# B&R Automation Studio project GAT (part 9)

#### CamAutomatActions.st
```iecst
//*********************************************************************************
//* Copyright: B&R Industrial Automation GmbH
//* Author:    B&R Industrial Automation GmbH
//* Created:   24 June, 2021/15:05
//* This task reads the cam automat data from the ACOPOS into the PV structure
//*********************************************************************************

ACTION InitCamAutFunctionBlocks:
	// Init cam automat related function blocks
	McCamAutDefine.DataAddress := ADR(McCamAutPar);
	MC_BR_CamAutomatGetPar_AcpAx_0.Slave := ADR(gAxisSlave);
	MC_BR_CamAutomatGetPar_AcpAx_0.Command := mcGET_PAR_ACTUAL;
	MC_BR_CamAutomatGetPar_AcpAx_0.CamAutomat := McCamAutDefine;
    MC_BR_CamAutomatSetPar_AcpAx_0.Command := mcSET_UPDATE_FROM_ADR;
    // Synchron means the new parameters are valid when an event with synchronous update = TRUE happens
	MC_BR_CamAutomatSetPar_AcpAx_0.AdvancedParameters.ParLock := mcCAMAUT_UNLOCK_SYNCHRON;
	MC_BR_CamAutomatSetPar_AcpAx_0.CamAutomat := McCamAutDefine;
	MC_BR_CamAutomatSetPar_AcpAx_0.Slave := ADR(gAxisSlave);
	MC_BR_CamAutomatCommand_0.Slave := ADR(gAxisSlave);
	MC_BR_CamAutomatCommand_0.Enable := TRUE;
END_ACTION

ACTION GetCamAutPar:
	CASE InitCamAut OF
		0: // Set up function blocks for reading and writing cam automat parameters
			MC_BR_CamAutomatGetPar_AcpAx_0.Execute := TRUE;
			InitCamAut := 1;

		1: // Wait for function block done
			IF MC_BR_CamAutomatGetPar_AcpAx_0.Done THEN
				MC_BR_CamAutomatGetPar_AcpAx_0.Execute := FALSE;
				InitCamAut := 10;
			END_IF
			// In case of error abort reading
			IF MC_BR_CamAutomatGetPar_AcpAx_0.Error THEN
				MC_BR_CamAutomatGetPar_AcpAx_0.Execute := FALSE;
				InitCamAut := 100;
			END_IF

		10: // Done, do nothing

		100: // Error handling
	END_CASE;
END_ACTION

ACTION UpdateCamAutomatAction:
	CASE CamUpdateState OF
		0: // Calculate new cam automat parameters
			IF UpdateCamAutomat AND (InitCamAut = 10) THEN
				// General CAM settings
				McCamAutPar.Common.Master.MasterStartInterval := MainCtrl.Intern.ProductLength[MainCtrl.Status.CurrentBatch];
				McCamAutPar.Common.Master.MasterStartPosition := 0;

				// CAM state 0: Base state, wait for master start position
				McCamAutPar.State[0].Event[0].NextState := 1;
				McCamAutPar.State[0].Event[0].SynchronousUpdate := mcSWITCH_ON;
                McCamAutPar.State[0].Event[0].Transition := mcEVENT_IMMEDIATELY;
                // Starts cutting process on interval, modify according to machine e.g. change to mcEVENT_SRC_TRIGGER1 for a signal wired to input channel 1 on ACOPOS
				McCamAutPar.State[0].Event[0].Type := mcEVENT_START_POSITION;

                // CAM state 1: First cut movement
                // * 100 because of measurement units to resolution units conversion
                McCamAutPar.State[1].MasterFactor := REAL_TO_DINT(GatDegreeToDistance(MainCtrl.FixParameter.SyncAngle, MainCtrl.FixParameter.CutDiameter / 2) * 100);
                // * 100 because of measurement units to resolution units conversion
                McCamAutPar.State[1].SlaveFactor := REAL_TO_DINT(MainCtrl.FixParameter.SyncAngle * 100);
                // Assuming print mark signals coincide with cutting positions
				McCamAutPar.State[1].CompensationParameters.MasterCompDistance := MainCtrl.Intern.ProductLength[MainCtrl.Status.CurrentBatch];
				IF MainCtrl.FixParameter.NrOfKnives = 0 THEN
					// There must be at least one knife!
					MainCtrl.FixParameter.NrOfKnives := 1;
				END_IF
				McCamAutPar.State[1].CompensationParameters.SlaveCompDistance := (360 / (2 * MainCtrl.FixParameter.NrOfKnives)) - (MainCtrl.FixParameter.SyncAngle / 2);
				// Change to next state at end of state
				McCamAutPar.State[1].Event[0].NextState := 3;
				McCamAutPar.State[1].Event[0].SynchronousUpdate := mcSWITCH_ON;
				McCamAutPar.State[1].Event[0].Transition := mcEVENT_END_OF_STATE;
				McCamAutPar.State[1].Event[0].Type := mcEVENT_SIGNAL2;
				McCamAutPar.State[1].Event[1].NextState := 2;
				McCamAutPar.State[1].Event[1].SynchronousUpdate := mcSWITCH_ON;
				McCamAutPar.State[1].Event[1].Transition := mcEVENT_END_OF_STATE;
				McCamAutPar.State[1].Event[1].Type := mcEVENT_STATE_END;

                // CAM state 2: Repeating cut movements
                // * 100 because of measurement units to resolution units conversion
				McCamAutPar.State[2].MasterFactor := REAL_TO_DINT(GatDegreeToDistance(MainCtrl.FixParameter.SyncAngle, MainCtrl.FixParameter.CutDiameter / 2) * 100);
				McCamAutPar.State[2].SlaveFactor := REAL_TO_DINT(MainCtrl.FixParameter.SyncAngle * 100);// * 100 because of measurement units to resolution units conversion
				McCamAutPar.State[2].CompensationParameters.MasterCompDistance := MainCtrl.Intern.ProductLength[MainCtrl.Status.CurrentBatch];
				McCamAutPar.State[2].CompensationParameters.SlaveCompDistance := (360 / MainCtrl.FixParameter.NrOfKnives);
				// Repeat state at end of state, or go to next state in case of signal 2 (stop cutting signal)
				McCamAutPar.State[2].Event[0].NextState := 3;
				McCamAutPar.State[2].Event[0].SynchronousUpdate := mcSWITCH_ON;
				McCamAutPar.State[2].Event[0].Transition := mcEVENT_END_OF_STATE;
				McCamAutPar.State[2].Event[0].Type := mcEVENT_SIGNAL2;
				McCamAutPar.State[2].Event[1].NextState := 2;
				McCamAutPar.State[2].Event[1].SynchronousUpdate := mcSWITCH_ON;
				McCamAutPar.State[2].Event[1].Transition := mcEVENT_END_OF_STATE;
				McCamAutPar.State[2].Event[1].Type := mcEVENT_STATE_END;

                // CAM state 3: Decelerate and stop at home position
                // Master with any positive value & slave = 0 means slave is not moving
                McCamAutPar.State[3].MasterFactor := 100;
                // Master with any positive value & slave = 0 means slave is not moving
                McCamAutPar.State[3].SlaveFactor := 0;
                // allow half a product length to stop
				McCamAutPar.State[3].CompensationParameters.MasterCompDistance := MainCtrl.Intern.ProductLength[MainCtrl.Status.CurrentBatch] / 2;
				McCamAutPar.State[3].CompensationParameters.SlaveCompDistance := (360 / (2 * MainCtrl.FixParameter.NrOfKnives));
				// Return to base state after axis has stopped
				McCamAutPar.State[3].Event[0].NextState := 0;
				McCamAutPar.State[3].Event[0].SynchronousUpdate := mcSWITCH_ON;
				McCamAutPar.State[3].Event[0].Transition := mcEVENT_END_OF_STATE;
				McCamAutPar.State[3].Event[0].Type := mcEVENT_STATE_END;

				MC_BR_CamAutomatSetPar_AcpAx_0.Execute := TRUE;
				CamUpdateState := 1;
			END_IF

		1: // Wait for SetPar done
			IF MC_BR_CamAutomatSetPar_AcpAx_0.Done THEN
				UpdateCamAutomat := FALSE;
				MC_BR_CamAutomatSetPar_AcpAx_0.Execute := FALSE;
				CamUpdateState := 0;
			ELSIF MC_BR_CamAutomatSetPar_AcpAx_0.Error THEN
				// Error handling
				MpAlarmXSet(gMpLinkAlarmXCore, 'SetCamFailed');
				UpdateCamAutomat := FALSE;
				MC_BR_CamAutomatSetPar_AcpAx_0.Execute := FALSE;
				CamUpdateState := 0;
			END_IF
	END_CASE;
END_ACTION
```

#### CrossCutter.st
```iecst
//*********************************************************************************
//* Copyright: B&R Industrial Automation GmbH
//* Created:   29 June, 2021/10:43
//* Process specific logic to update production information and process parameters
//*********************************************************************************

ACTION CrossCutter:

	//****************************Starting and stopping the process*********************************
    IF MainCtrl.Command.AutoModeOn THEN
        // Switch on axes
		AxisControl[AXIS_IDX_FEEDER].Command.Power := TRUE;
		AxisControl[AXIS_IDX_CUTTER].Command.Power := TRUE;
		// Home axes if not homed yet
		IF NOT MpAxisBasic_x[AXIS_IDX_FEEDER].IsHomed AND (AxisControl[AXIS_IDX_FEEDER].AxisState = AX_STATE_WAIT) THEN
			AxisControl[AXIS_IDX_FEEDER].Command.Home := TRUE;
		END_IF
		IF NOT MpAxisBasic_x[AXIS_IDX_CUTTER].IsHomed AND (AxisControl[AXIS_IDX_CUTTER].AxisState = AX_STATE_WAIT) THEN
			AxisControl[AXIS_IDX_CUTTER].Command.Home := TRUE;
		END_IF

		// Reset run switches when in error state
		IF (AxisControl[AXIS_IDX_FEEDER].AxisState = AX_STATE_ERROR) OR (AxisControl[AXIS_IDX_CUTTER].AxisState = AX_STATE_ERROR) THEN
			MainCtrl.Command.RunCutter := FALSE;
			MainCtrl.Command.RunFeeder := FALSE;
		END_IF

		// Start movement of feeder axis
		AxisControl[AXIS_IDX_FEEDER].Command.MoveVelocity := MainCtrl.Command.RunFeeder;

		// Start synchronized movement of Cutter with cam automat
		IF MainCtrl.Command.RunCutter THEN
			AxisControl[AXIS_IDX_CUTTER].Command.RunCamAutomat := TRUE;
		ELSE
			// If axis is moving use signal1 to stop slave in home position after the current product is done, otherwise stop now
			IF (MpAxisBasic_x[AXIS_IDX_CUTTER].Velocity > 0) AND MC_BR_CamAutomatCommand_0.Running THEN
				MC_BR_CamAutomatCommand_0.SetSignal1 := TRUE;
			ELSE
				// Back in base state reset signal and end camautomat
				MC_BR_CamAutomatCommand_0.SetSignal1 := FALSE;
				MC_BR_CamAutomatCommand_0.EndAutomat := MC_BR_CamAutomatCommand_0.Running;
				IF NOT MC_BR_CamAutomatCommand_0.Running THEN
					// Automat has stopped
					AxisControl[AXIS_IDX_CUTTER].Command.RunCamAutomat := FALSE;
				END_IF
			END_IF
		END_IF
	ELSIF LastAutoModeOn THEN
		// Auto mode is switched off, reste run commands
		MainCtrl.Command.RunCutter := FALSE;
		AxisControl[AXIS_IDX_CUTTER].Command.RunCamAutomat := FALSE;
		MainCtrl.Command.RunFeeder := FALSE;
		AxisControl[AXIS_IDX_FEEDER].Command.MoveVelocity := FALSE;
	END_IF
	LastAutoModeOn := MainCtrl.Command.AutoModeOn;

	//********************************Parameters Limits************

	IF (AxisControl[AXIS_IDX_FEEDER].Parameter.AxPar.Velocity = 0) AND AxisControl[AXIS_IDX_FEEDER].Command.MoveVelocity THEN
		MpAlarmXSet(gMpLinkAlarmXCore, 'FeederSpeedNotSet');
		AxisControl[AXIS_IDX_FEEDER].Command.MoveVelocity := FALSE;
	END_IF
	IF (AxisControl[AXIS_IDX_CUTTER].Parameter.AxPar.Velocity = 0) AND AxisControl[AXIS_IDX_CUTTER].Command.MoveAdditive THEN
		MpAlarmXSet(gMpLinkAlarmXCore, 'CutterSpeedNotSet');
		AxisControl[AXIS_IDX_CUTTER].Command.MoveAdditive := FALSE;
	END_IF
	IF (AxisControl[AXIS_IDX_CUTTER].Parameter.AxPar.Distance = 0) AND (AxisControl[AXIS_IDX_CUTTER].Command.MoveAdditive)  THEN
		MpAlarmXSet(gMpLinkAlarmXCore, 'CutterPositionNotSet');
		AxisControl[AXIS_IDX_CUTTER].Command.MoveAdditive := FALSE;
	END_IF

	//****************************Product Cutting numbering*********************************
    // Update parameters on recipe load
    IF MpRecipeRegPar_P.UpdateNotification THEN
		brsmemcpy(ADR(MainCtrl.Intern.ProductLength), ADR(MainCtrl.Parameter.ProductLength), SIZEOF(MainCtrl.Intern.ProductLength));
		brsmemcpy(ADR(MainCtrl.Intern.ProductNumber), ADR(MainCtrl.Parameter.ProductNumber), SIZEOF(MainCtrl.Intern.ProductNumber));
		UpdateCamAutomat := TRUE;
	END_IF

	// InCam -> next cut is starting
	IF EDGEPOS(MC_BR_CamAutomatCommand_0.InCam) THEN
		MainCtrl.Status.ProductsCutBatch := MainCtrl.Status.ProductsCutBatch + 1;
		MainCtrl.Status.ProductsCutTotal := MainCtrl.Status.ProductsCutTotal + 1;
	END_IF

	// Batch finished, start next batch -> adjust cam automat parameters for next batches product length
	IF (MainCtrl.Status.ProductsCutBatch >= MainCtrl.Intern.ProductNumber[MainCtrl.Status.CurrentBatch])
		AND (MainCtrl.Status.ProductsCutBatch > 0) THEN
		// Set new cam automat values
		MainCtrl.Status.CurrentBatch := MainCtrl.Status.CurrentBatch + 1;
		IF MainCtrl.Status.CurrentBatch > 4 THEN
			MainCtrl.Status.CurrentBatch := 0;
		END_IF
		MainCtrl.Status.ProductsCutBatch := 0;
		UpdateCamAutomat := TRUE;
	END_IF
	MainCtrl.Status.CurrentBatchTarget := MainCtrl.Intern.ProductNumber[MainCtrl.Status.CurrentBatch];
	MainCtrl.Status.CurrentBatchLength := MainCtrl.Intern.ProductLength[MainCtrl.Status.CurrentBatch];

	// Action to handle cam automat updates
	UpdateCamAutomatAction;

END_ACTION
```

#### Main.st
```iecst
//*********************************************************************************
//* Copyright: B&R Industrial Automation GmbH
//* Author:    B&R Industrial Automation GmbH
//* Created:   30. Sep 2020/08:00
//* Description: Tasks for axis control. The Main Cross Cutter handling is done in this task.
//*********************************************************************************

PROGRAM _INIT
	// Register parameters to MpRecipe
	MpRecipeRegPar_M.MpLink := ADR(gMpLinkRecipeXml);
	MpRecipeRegPar_M.Enable := TRUE;
	MpRecipeRegPar_M.Category := ADR('Machine');
	MpRecipeRegPar_M.PVName := ADR('MainCtrl:MainCtrl.FixPar');
	MpRecipeRegPar_P.MpLink := ADR(gMpLinkRecipeXml);
	MpRecipeRegPar_P.Enable := TRUE;
	MpRecipeRegPar_P.Category := ADR('Parameters');
	MpRecipeRegPar_P.PVName := ADR('MainCtrl:MainCtrl.Para');
	MpRecipeRegPar_Pre1.MpLink := ADR(gRecipeXmlPreviewMpLink);
	MpRecipeRegPar_Pre1.Enable := TRUE;
	MpRecipeRegPar_Pre1.Category := ADR('Preview');
	MpRecipeRegPar_Pre1.PVName := ADR('MainCtrl:PreviewParameters');
	MpRecipeRegPar_Pre2.MpLink := ADR(gMpLinkRecipeXml);
	MpRecipeRegPar_Pre2.Enable := TRUE;
	MpRecipeRegPar_Pre2.Category := ADR('Parameters');
	MpRecipeRegPar_Pre2.PVName := ADR('MainCtrl:PreviewParameters');

	// Activate RegPar FUBs
	WHILE NOT MpRecipeRegPar_M.Active DO
		MpRecipeRegPar_M();
	END_WHILE
	WHILE NOT MpRecipeRegPar_P.Active DO
		MpRecipeRegPar_P();
	END_WHILE
	WHILE NOT MpRecipeRegPar_Pre1.Active DO
		MpRecipeRegPar_Pre1();
	END_WHILE
    WHILE NOT MpRecipeRegPar_Pre2.Active DO
		MpRecipeRegPar_Pre2();
	END_WHILE

    // Init Cam automat related function blocks ***************************************
	InitCamAutFunctionBlocks;

	// Axis No.0 initialization *********************************************************************************
	MpAxisBasic_x[0].MpLink := ADR(gAxisMaster);
	MpAxisBasic_x[0].Enable := TRUE;
	MpAxisBasic_x[0].Parameters := ADR(AxisControl[0].Parameter.AxPar);
	MC_ReadAxisError_x[0].Axis := ADR(gAxisMaster);
	MC_ReadActualTorque_x[0].Axis := ADR(gAxisMaster);

	// Axis No.1 initialization *********************************************************************************
	MpAxisBasic_x[1].MpLink := ADR(gAxisSlave);
	MpAxisBasic_x[1].Enable := TRUE;
	MpAxisBasic_x[1].Parameters := ADR(AxisControl[1].Parameter.AxPar);
	MC_ReadAxisError_x[1].Axis := ADR(gAxisSlave);
	MC_ReadActualTorque_x[1].Axis := ADR(gAxisSlave);
END_PROGRAM

PROGRAM _CYCLIC

	//******************** Init cam automat parameters ********************
	GetCamAutPar;

	//******************** Axis status updates ********************
	//******************** Status information is read before the state machine to attain a shorter reaction time in case of error ********************
	AxisStatusUpdate;

	//******************** Axis control ********************
	AxisStateMachine;

	//******************** Crosscutter control ********************
	CrossCutter;

	//*************************************************

	//******************** Copy preview parameters before creating or saving a recipe ********************
	IF CopyPreviewParameters THEN
		PreviewParameters := MainCtrl.Parameter;
		CopyPreviewParameters := FALSE;
	END_IF
	IF ResetEditValues THEN
		MainCtrl.Parameter := PreviewParameters;
		ResetEditValues := FALSE;
    END_IF

	//******************** MpAxisBasic function block calls ********************
	FOR AxIndex := 0 TO MAX_IDX_AXIS DO
		MpAxisBasic_x[AxIndex]();
	END_FOR

	//******************** CamAutomat function block calls ********************
	MC_BR_CamAutomatSetPar_AcpAx_0();
	MC_BR_CamAutomatGetPar_AcpAx_0();
	MC_BR_CamAutomatCommand_0();

	//******************** MpRecipeRegPar FB calls ********************
	MpRecipeRegPar_M();
	MpRecipeRegPar_P();
	MpRecipeRegPar_Pre1();
	MpRecipeRegPar_Pre2();
END_PROGRAM

PROGRAM _EXIT
	MpRecipeRegPar_M.Enable := FALSE;
	MpRecipeRegPar_M();
	MpRecipeRegPar_P.Enable := FALSE;
	MpRecipeRegPar_P();
	MpRecipeRegPar_Pre1.Enable := FALSE;
	MpRecipeRegPar_Pre1();
	MpRecipeRegPar_Pre2.Enable := FALSE;
	MpRecipeRegPar_Pre2();
	FOR AxIndex := 0 TO MAX_IDX_AXIS DO
		MpAxisBasic_x[AxIndex].Enable := FALSE;
		MpAxisBasic_x[AxIndex]();
	END_FOR
END_PROGRAM
```

### Program Logical/MainControl/PIDControl

#### Types.typ
```iecst
TYPE
	PidState_enum :
		(
		PID_IDLE := 0,
		PID_ACTIVE := 1,
		PID_TUNING := 2,
		PID_ERROR := 3
		);
	PidControlParameters_type : 	STRUCT
		PidParameters : MTPIDParametersType;
		SetValue : REAL;
		MinOut : REAL;
		MaxOut : REAL;
		Invert : BOOL;
	END_STRUCT;
END_TYPE
```

#### Variables.var
```iecst
VAR
	MTBasicsPID_0 : MTBasicsPID; (*Pid control function block*)
	MpRecipeRegPar_Pre : MpRecipeRegPar; (*Register parameters for preview function*)
	MpRecipeRegPar_P : MpRecipeRegPar; (*Register parameters in the recipe*)
	PidControlParameters : PidControlParametersType; (*Pid parameters*)
	SimAddValue : REAL; (*Simulated add value*)
	OutValue : REAL; (*out value*)
	ActValue : REAL; (*actual value*)
	SimulationActive : BOOL; (*simulation on/off*)
	MTBasicsOscillationTuning_0 : MTBasicsOscillationTuning; (*Oscillation tuning function block*)
	TuningQuality : REAL; (*Tuning quality in percent*)
	PidStatus : PidStateEnum; (*Pid status value used for the status snippet*)
END_VAR
```

#### Main.st
```iecst
//*********************************************************************************
//* Copyright: B&R Industrial Automation GmbH
//* Created:   22 July, 2021/15:54
//* This task contains the logic for a PID controller
//*********************************************************************************

PROGRAM _INIT
	// Register parameters to the recipe
	MpRecipeRegPar_P.MpLink := ADR(gMpLinkRecipeXml);
	MpRecipeRegPar_P.Enable := TRUE;
	MpRecipeRegPar_P.PVName := ADR('PIDControl:PidControlParameters');
	MpRecipeRegPar_P.Category := ADR('Product');
	MpRecipeRegPar_Pre.MpLink := ADR(gRecipeXmlPreviewMpLink);
	MpRecipeRegPar_Pre.Enable := TRUE;
	MpRecipeRegPar_Pre.PVName := ADR('PIDControl:PidControlParameters');
	MpRecipeRegPar_Pre.Category := ADR('Preview');
	// Activate recipe registration
	WHILE NOT MpRecipeRegPar_P.Active DO
		MpRecipeRegPar_P();
	END_WHILE
	WHILE NOT MpRecipeRegPar_Pre.Active DO
		MpRecipeRegPar_Pre();
	END_WHILE
	// Keep start signal of tuning fub true, tuning is started and stopped via HMI by setting the enable input
	MTBasicsOscillationTuning_0.Start := TRUE;
END_PROGRAM

PROGRAM _CYCLIC
	// Simulation
	SimulateActValue;

	// Update parameters on update notification
	IF MpRecipeRegPar_P.UpdateNotification THEN
		MTBasicsPID_0.PIDParameters := PidControlParameters.PidParameters;
		MTBasicsPID_0.SetValue := PidControlParameters.SetValue;
		MTBasicsPID_0.MinOut := PidControlParameters.MinOut;
		MTBasicsPID_0.MaxOut := PidControlParameters.MaxOut;
		MTBasicsPID_0.Invert := PidControlParameters.Invert;
		MTBasicsPID_0.Update := MTBasicsPID_0.Active;
		MTBasicsOscillationTuning_0.MinOut := PidControlParameters.MinOut;
		MTBasicsOscillationTuning_0.MaxOut := PidControlParameters.MaxOut;
		MTBasicsOscillationTuning_0.SetValue := PidControlParameters.SetValue;
		MTBasicsOscillationTuning_0.Invert := PidControlParameters.Invert;
		MTBasicsOscillationTuning_0.Update := MTBasicsOscillationTuning_0.Active;
	END_IF

	// Update actual value
	MTBasicsPID_0.ActValue := ActValue;
	MTBasicsOscillationTuning_0.ActValue := ActValue;

	// Autotuning of parameters
	IF MTBasicsOscillationTuning_0.TuningDone THEN
		PidControlParameters.PidParameters := MTBasicsOscillationTuning_0.PIDParameters;
		TuningQuality := MTBasicsOscillationTuning_0.Quality;
	END_IF

	// Reset update commands
	IF MTBasicsPID_0.UpdateDone THEN
		MTBasicsPID_0.Update := FALSE;
	ELSIF MTBasicsOscillationTuning_0.UpdateDone THEN
		MTBasicsOscillationTuning_0.Update := FALSE;
	END_IF

	// Call function blocks
	MpRecipeRegPar_P();
	MpRecipeRegPar_Pre();
	MTBasicsPID_0();
	MTBasicsOscillationTuning_0();

	// Update status value
	IF MTBasicsOscillationTuning_0.TuningActive THEN
		PidStatus := PID_TUNING;
	ELSIF MTBasicsPID_0.Error THEN
		PidStatus := PID_ERROR;
	ELSIF MTBasicsPID_0.Active THEN
		PidStatus := PID_ACTIVE;
	ELSE
		PidStatus := PID_IDLE;
	END_IF

	// Set output value
	IF MTBasicsOscillationTuning_0.TuningActive THEN
		OutValue := MTBasicsOscillationTuning_0.Out;
	ELSE
		OutValue := MTBasicsPID_0.Out;
	END_IF
END_PROGRAM

PROGRAM _EXIT
	MpRecipeRegPar_P.Enable := FALSE;
	MpRecipeRegPar_P();
	MpRecipeRegPar_Pre.Enable := FALSE;
	MpRecipeRegPar_Pre();
END_PROGRAM
```

#### SimulateActValue.st
```iecst
//*********************************************************************************
//* Copyright: B&R Industrial Automation GmbH
//* Created:   23 July, 2021/08:47
//* Simulation of the actual value
//*********************************************************************************
ACTION SimulateActValue:
	IF SimulationActive THEN
		SimAddValue := (SimAddValue * 0.99) + (OutValue * 0.01);
		ActValue := (ActValue * 0.9999) + (0.01 * SimAddValue);
	END_IF
END_ACTION
```

### Package Logical/MachineControl - Package for Machine Control

### Package Logical/MachineControl/AxisTemplate - Package for mapp Axis Framework Template

### Program Logical/MachineControl/AxisTemplate/AxisMgr

#### AxisMgr.typ
```iecst
(*Structure types*)

TYPE
	AxisSettingsType : 	STRUCT
		AxisFeatures : {REDUND_UNREPLICABLE} ARRAY[0..2]OF STRING[255]; (*Variable to write axis features into*)
		DriveConfiguration : {REDUND_UNREPLICABLE} McCfgPureVAxType; (*Drive configuration structure*)
		BaseConfiguration : {REDUND_UNREPLICABLE} McCfgAxType; (*Base axis type configuration *)
		BaseParam : {REDUND_UNREPLICABLE} McCfgAxMoveLimType; (*Base axis movement configuration*)
	END_STRUCT;
	AxisMachineSettingsType : {REDUND_UNREPLICABLE} 	STRUCT
		ReferencePosition : {REDUND_UNREPLICABLE} LREAL := 0; (*[mm] Axis position after reference*)
	END_STRUCT;
	AxisControlCommandType : {REDUND_UNREPLICABLE} 	STRUCT
		UpdatePreviewParameters : {REDUND_UNREPLICABLE} BOOL; (*Cmd to load new preview*)
		LoadRecipeParameters : {REDUND_UNREPLICABLE} BOOL; (*Load selected recipe file into active parameters *)
		SaveRecipeParameters : {REDUND_UNREPLICABLE} BOOL; (*Save current parameters*)
		Power : {REDUND_UNREPLICABLE} BOOL; (*Cmd power*)
		Reference : {REDUND_UNREPLICABLE} BOOL; (*Cmd home / reference*)
		MoveAbsolute : {REDUND_UNREPLICABLE} BOOL; (*Cmd move absolute*)
		MoveAdditive : {REDUND_UNREPLICABLE} BOOL; (*Cmd move additive*)
		MoveToStart : {REDUND_UNREPLICABLE} BOOL; (*Cmd move the start position*)
		Abort : {REDUND_UNREPLICABLE} BOOL; (*Cmd abort*)
		Stop : {REDUND_UNREPLICABLE} BOOL; (*Cmd stop all movement*)
		Reset : {REDUND_UNREPLICABLE} BOOL; (*Cmd reset axis state*)
		JogPositive : {REDUND_UNREPLICABLE} BOOL; (*Cmd jog positive*)
		JogNegative : {REDUND_UNREPLICABLE} BOOL; (*Cmd jog negative*)
		Start : {REDUND_UNREPLICABLE} BOOL; (*Cmd start motion*)
	END_STRUCT;
	AxisControlParametersType : {REDUND_UNREPLICABLE} 	STRUCT
		HomePosition : {REDUND_UNREPLICABLE} LREAL := 0; (*[mm] Home Position*)
		Position : {REDUND_UNREPLICABLE} LREAL := 0; (*[mm] Position for absolute move*)
		Distance : {REDUND_UNREPLICABLE} LREAL := 50; (*[mm] Distance for relative move*)
		Velocity : {REDUND_UNREPLICABLE} REAL := 100; (*[mm/s] Velocity for absoluate and relative moves*)
		Acceleration : {REDUND_UNREPLICABLE} REAL := 360; (*[mm/s2] Acceleration for absoluate and relative moves*)
		Deceleration : {REDUND_UNREPLICABLE} REAL := 360; (*[mm/s2] Deceleration for absoluate and relative moves*)
		JogVelocity : {REDUND_UNREPLICABLE} REAL := 100; (*[mm/s] Velocity used when jogging the axis*)
		StopDeceleration : {REDUND_UNREPLICABLE} REAL := 720; (*[mm/s2] Deceleration for stopping*)
	END_STRUCT;
	AxisControlStatusType : {REDUND_UNREPLICABLE} 	STRUCT
		TaskName : {REDUND_UNREPLICABLE} STRING[80]; (*Current task name for configuration changes*)
		MachineSettingsName : {REDUND_UNREPLICABLE} STRING[255]; (*Category name for machine settings*)
		ProductSettingsName : {REDUND_UNREPLICABLE} STRING[255]; (*Category name for product settings*)
		Status : {REDUND_UNREPLICABLE} STRING[80]; (*Machine Status*)
		IsReady : {REDUND_UNREPLICABLE} BOOL; (*Axis is ready*)
		ErrorActive : {REDUND_UNREPLICABLE} BOOL; (*Error active*)
		Busy : {REDUND_UNREPLICABLE} BOOL; (*Cmd execution*)
		ReferenceRequired : {REDUND_UNREPLICABLE} BOOL; (*Reference cmd required*)
		Position : {REDUND_UNREPLICABLE} LREAL; (*Current position*)
		Velocity : {REDUND_UNREPLICABLE} REAL; (*Current position*)
		Current : {REDUND_UNREPLICABLE} REAL; (*Drive current*)
		LagError : {REDUND_UNREPLICABLE} LREAL; (*Axis lag error *)
		MotorTemperature : {REDUND_UNREPLICABLE} REAL; (*Motor temperature*)
		IsHomed : {REDUND_UNREPLICABLE} BOOL; (*Axis is referenced*)
		IsPowered : {REDUND_UNREPLICABLE} BOOL; (*Axis is powered*)
	END_STRUCT;
	AxisControlType : {REDUND_UNREPLICABLE} 	STRUCT
		Command : {REDUND_UNREPLICABLE} AxisControlCommandType; (*Cmd structure*)
		Parameters : {REDUND_UNREPLICABLE} AxisControlParametersType; (*Parameter structure*)
		Status : {REDUND_UNREPLICABLE} AxisControlStatusType; (*Status structure*)
	END_STRUCT;
	AxisRecipeType : 	STRUCT
		EditDialogOpened : BOOL; (*HMI edit dialog open*)
		CreateDialogOpened : BOOL; (*HMI create dialog open*)
		SaveRecipe : BOOL; (*Cmd save current values*)
		LoadRecipe : BOOL; (*Cmd load exiting recipe*)
		CreateRecipe : BOOL; (*Cmd create new recipe*)
		State : AxisRecipeStepEnum; (*Recipe handling state*)
		CategoryDropdown : STRING[50]; (*HMI selector*)
	END_STRUCT;
END_TYPE

(*Enumerations*)

TYPE
	StateEnum :
		(
		STATE_INIT, (*Axis initialization state*)
		STATE_POWER_ON, (*Axis powering on state*)
		STATE_HOME, (*Axis homing state*)
		STATE_REFERENCE, (*Axis reference state*)
		STATE_MOVE_TO_HOME_POSITION, (*Axis moving to reference position state*)
		STATE_READY, (*Axis ready state*)
		STATE_MANUAL_OPERATION, (*Axis manual state*)
		STATE_AUTOMATIC_OPERATION, (*Axis automatic state*)
		STATE_STOPPING, (*Axis stopping state*)
		STATE_STOPPED, (*Axis stopped state*)
		STATE_ABORTING, (*Axis aborting state*)
		STATE_ABORTED, (*Axis aborted state*)
		STATE_CLEARING, (*Axis clearing state*)
		STATE_RESETTING (*Axis resetting state*)
		);
	ParameterStateEnum :
		(
		PAR_STATE_INIT, (*Param initialization state*)
		PAR_STATE_READ, (*Param read state*)
		PAR_STATE_WRITE, (*Param write state*)
		PAR_STATE_READY (*Param ready state*)
		);
	ConfigurationStateEnum :
		(
		CONFIG_STATE_INIT, (*Config initialization state*)
		CONFIG_STATE_READ, (*Config read state*)
		CONFIG_STATE_WRITE, (*Config write state*)
		CONFIG_STATE_READY (*Config ready state*)
		);
	ManualStateEnum :
		(
		MANUAL_STATE_IDLE, (*Idle state*)
		MANUAL_STATE_JOG, (*Jog state*)
		MANUAL_STATE_MOVE, (*Move state*)
		MANUAL_STATE_STOPPING (*Stopping state*)
		);
	AutomaticStateEnum :
		(
		AUTOMATIC_STATE_IDLE, (*Idle state*)
		AUTOMATIC_STATE_RUNNING (*Run state*)
		);
	AxisRecipeStepEnum :
		(
		REC_AXIS_WAIT, (*Wait state*)
		REC_AXIS_LOAD, (*Load product parameters*)
		REC_AXIS_SAVE, (*Save product parameters*)
		REC_AXIS_CREATE, (*Create new axis recipe*)
		REC_AXIS_STORE_MACH_SETTINGS, (*Save machine parameter settings*)
		REC_AXIS_FACTORY_RESET (*Factory reset*)
		);
END_TYPE
```

#### AxisMgr.var
```iecst
VAR
	i : {REDUND_UNREPLICABLE} USINT; (*Loop index variable*)
	ParameterState : {REDUND_UNREPLICABLE} ParameterStateEnum; (*Parameter handling state*)
	ConfigurationState : {REDUND_UNREPLICABLE} ConfigurationStateEnum; (*Configuration handling state*)
	State : {REDUND_UNREPLICABLE} StateEnum; (*OMAC based state machine*)
	AutomaticState : {REDUND_UNREPLICABLE} AutomaticStateEnum; (*Automatic handling state*)
	ManualState : {REDUND_UNREPLICABLE} ManualStateEnum; (*Manual handling state*)
	AxisControl : {REDUND_UNREPLICABLE} AxisControlType; (*Single axis control type*)
	AxisSettings : {REDUND_UNREPLICABLE} AxisSettingsType; (*Single axis settings *)
END_VAR
(*Function Blocks*)
VAR
	MC_BR_CheckRestorePositionData_0 : {REDUND_UNREPLICABLE} MC_BR_CheckRestorePositionData; (*Check restore postion data*)
	RestorePosition : {REDUND_UNREPLICABLE} McAcpAxRestorePosType; (*Data structure for retsore position mode*)
	MpRecipeRegPar_Cfg : {REDUND_UNREPLICABLE} MpRecipeRegPar; (*Register function block for configuration values*)
	MpRecipeRegPar_Par : {REDUND_UNREPLICABLE} MpRecipeRegPar; (*Register function block for parameter values*)
	MpAlarmXCore_0 : {REDUND_UNREPLICABLE} MpAlarmXCore; (*AlarmX Core function block*)
	MpAxisParameters : {REDUND_UNREPLICABLE} MpAxisBasicParType := (Distance:=70,Velocity:=100,Acceleration:=5000,Deceleration:=5000,Jog:=(Velocity:=70,Acceleration:=5000,Deceleration:=5000),AutoTune:=(MaxCurrentPercent:=50,MaxDistance:=720,MaxPositionError:=5)); (*Standard MpAxis parameter structure *)
	MpAxisBasic_0 : {REDUND_UNREPLICABLE} MpAxisBasic; (*MpAxis main function block*)
	MC_BR_ProcessConfig_AX : {REDUND_UNREPLICABLE} MC_BR_ProcessConfig; (*Function block to read and write the axis configuration*)
	MC_BR_ProcessConfig_ACP : {REDUND_UNREPLICABLE} MC_BR_ProcessConfig; (*Function block to read and write the ACOPOS configuration*)
	IsHomedEdgePos : {REDUND_UNREPLICABLE} R_TRIG; (*Detecting rising edge for Homed*)
	InPositionEdgePos : {REDUND_UNREPLICABLE} R_TRIG; (*Detecting rising edge for InPosition*)
	ReferenceEdgePos : {REDUND_UNREPLICABLE} R_TRIG; (*Detecting rising edge for Referenced*)
	MC_BR_ProcessParam_AX : {REDUND_UNREPLICABLE} MC_BR_ProcessParam; (*Function block to read and write the ACOPOS parameters*)
	MpAlarmXControl_SpeedNotSet : MpAlarmXAlarmControl; (*AlarmX control function block*)
END_VAR
(*Recipe*)
VAR
	ParametersEdit : {REDUND_UNREPLICABLE} AxisControlParametersType; (*Parameter structure used in recipe for edit*)
	ParametersPreview : {REDUND_UNREPLICABLE} AxisControlParametersType; (*Parameter structure used in recipe for preview*)
	MachineSettings : {REDUND_UNREPLICABLE} AxisMachineSettingsType; (*Machine settings structure*)
	MachineSettingsEdit : {REDUND_UNREPLICABLE} AxisMachineSettingsType; (*Machine settings structure used in recipe for edit*)
	MachineSettingsPreview : {REDUND_UNREPLICABLE} AxisMachineSettingsType; (*Machine settings structure used in recipe for preview*)
	AxisRecipe : {REDUND_UNREPLICABLE} AxisRecipeType; (*HMI interface structure*)
END_VAR
```

#### AutomaticCommand.st
```iecst
// Returns True if an automatic command is active
FUNCTION AutomaticCommand

    AutomaticCommand := Commands.Start;

END_FUNCTION
```

#### AxisControlModes.st
```iecst
ACTION AxisInit:

END_ACTION

ACTION AxisCyclic:

    IF (MpRecipeRegPar_Par.UpdateNotification) THEN

    END_IF

END_ACTION

ACTION AxisManual:

    MpAxisParameters.Jog.Velocity := AxisControl.Parameters.JogVelocity;
    MpAxisParameters.Position := AxisControl.Parameters.Position;
    MpAxisParameters.Distance := AxisControl.Parameters.Distance;
    MpAxisParameters.Acceleration := AxisControl.Parameters.Acceleration;
    MpAxisParameters.Deceleration := AxisControl.Parameters.Deceleration;

    CASE ManualState OF
        MANUAL_STATE_IDLE:
            IF ((AxisControl.Command.JogNegative = TRUE) OR (AxisControl.Command.JogPositive = TRUE)) THEN
                ManualState := MANUAL_STATE_JOG;
            ELSIF ((AxisControl.Command.MoveAbsolute = TRUE) OR (AxisControl.Command.MoveAdditive = TRUE)) THEN
                MpAxisBasic_0.MoveAbsolute := AxisControl.Command.MoveAbsolute;
                MpAxisBasic_0.MoveAdditive := AxisControl.Command.MoveAdditive;
                AxisControl.Command.MoveAbsolute := FALSE;
                AxisControl.Command.MoveAdditive := FALSE;
                ManualState := MANUAL_STATE_MOVE;
            END_IF

        MANUAL_STATE_JOG:
            MpAxisBasic_0.JogNegative := AxisControl.Command.JogNegative;
            MpAxisBasic_0.JogPositive := AxisControl.Command.JogPositive;
            IF (AxisControl.Command.Stop = TRUE) THEN
                AxisControl.Command.Stop := FALSE;
                MpAxisBasic_0.Stop := TRUE;
                ManualState := MANUAL_STATE_STOPPING;
            ELSIF ((AxisControl.Command.JogNegative = FALSE) AND (AxisControl.Command.JogPositive = FALSE)) THEN
                MpAxisBasic_0.Stop := FALSE;
                MpAxisBasic_0.JogPositive := FALSE;
                MpAxisBasic_0.JogNegative := FALSE;
                ManualState := MANUAL_STATE_STOPPING;
            END_IF

        MANUAL_STATE_MOVE:
            IF (AxisControl.Command.Stop = TRUE) THEN
                MpAxisBasic_0.MoveAbsolute := FALSE;
                MpAxisBasic_0.MoveAdditive := FALSE;
                AxisControl.Command.Stop := FALSE;
                MpAxisBasic_0.Stop := TRUE;
                ManualState := MANUAL_STATE_STOPPING;
            ELSIF (InPositionEdgePos.Q = TRUE) THEN
                MpAxisBasic_0.MoveAbsolute := FALSE;
                MpAxisBasic_0.MoveAdditive := FALSE;
                ManualState := MANUAL_STATE_IDLE;
                state := STATE_READY;
            ELSIF ((AxisControl.Command.JogNegative = TRUE) OR (AxisControl.Command.JogPositive = TRUE)) THEN
                MpAxisBasic_0.MoveAbsolute := FALSE;
                MpAxisBasic_0.MoveAdditive := FALSE;
                ManualState := MANUAL_STATE_JOG;
            END_IF

        MANUAL_STATE_STOPPING:
            MpAxisBasic_0.JogNegative := FALSE;
            MpAxisBasic_0.JogPositive := FALSE;
            MpAxisBasic_0.MoveAbsolute := FALSE;
            MpAxisBasic_0.MoveAdditive := FALSE;

            IF (MpAxisBasic_0.MoveActive = FALSE) THEN
                ManualState := MANUAL_STATE_IDLE;
                state := STATE_READY;
            END_IF
    END_CASE

END_ACTION

ACTION AxisAutomatic:

    CASE AutomaticState OF
        AUTOMATIC_STATE_IDLE:
            IF (AxisControl.Command.Start = TRUE) THEN
                MpAlarmXControl_SpeedNotSet.Set := (MpAxisParameters.Velocity = 0);
                AxisControl.Command.Start := FALSE;
                AutomaticState := AUTOMATIC_STATE_RUNNING;
            END_IF

        AUTOMATIC_STATE_RUNNING:
            MpAxisBasic_0.MoveVelocity := TRUE;
            MpAxisParameters.Velocity := AxisControl.Parameters.Velocity;
            MpAxisParameters.Acceleration := AxisControl.Parameters.Acceleration;
            MpAxisParameters.Deceleration := AxisControl.Parameters.Deceleration;

            IF (AxisControl.Command.Stop = TRUE) THEN
                AxisControl.Command.Stop := FALSE;
                MpAxisBasic_0.MoveVelocity := FALSE;
                state := STATE_READY;
                AutomaticState := AUTOMATIC_STATE_IDLE;
            END_IF
    END_CASE

END_ACTION

ACTION AxisReset:

END_ACTION
```

#### AxisMgr.st
```iecst
//***********************************************************************
// Copyright: B&R Industrial Automation GmbH
// Author: B&R Industrial Automation GmbH
// Created: Jan 1, 2022
// Description: Tasks for axis control.
//***********************************************************************

PROGRAM _INIT
    // Read current task name for category setup
    ST_name(0, ADR(AxisControl.Status.TaskName), 0);

	// Inititialize mapp function blocks
	MpAlarmXCore_0.Enable := TRUE;
	MpAlarmXCore_0();
    ConfigurationInit;

    MpAxisBasic_0.Enable := TRUE;
	MpAxisBasic_0.MpLink := ADR(gAxisTemplate);
	MpAxisBasic_0();

    AxisInit;

END_PROGRAM

PROGRAM _CYCLIC

    MpAxisBasic_0.MpLink := ADR(gAxisTemplate);
    MC_BR_CheckRestorePositionData_0.Axis := ADR(gAxisTemplate);

	// Call all actions
    SimulationControl;
    AxisStateMachine;
    AxisCyclic;
	RecipeCyclic;

    // Assign MpLink
    MpAlarmXCore_0.MpLink := ADR(gAlarmXCore_AxisTemplate);

	// Call function block
	MpAlarmXCore_0();

END_PROGRAM

PROGRAM _EXIT

	// Disable the function blocls to unlink the MpLinks.
	// Do NOT disable MpAxisBasic, as this can cause problems during project transfer.
    MpRecipeRegPar_Par.Enable := FALSE;
	MpRecipeRegPar_Cfg.Enable := FALSE;
	MpAlarmXCore_0.Enable := FALSE;

	// Call function blocks
	MpRecipeRegPar_Par();
	MpRecipeRegPar_Cfg();
	MpAlarmXCore_0();

END_PROGRAM
```

#### ManualCommand.st
```iecst
// Returns True if a manual command is active, false otherwise
FUNCTION ManualCommand

	ManualCommand := Commands.JogNegative OR Commands.JogPositive OR Commands.MoveAbsolute OR Commands.MoveAdditive;

END_FUNCTION
```

#### Recipe.st
```iecst
ACTION RecipeInit:

    // Register the variables with the recipe system
    AxisControl.Status.ProductSettingsName := AxisControl.Status.TaskName;
    brsstrcat(ADR(AxisControl.Status.ProductSettingsName), ADR(':ParametersPreview'));
    MpRecipeRegPar_Par.MpLink := ADR(gMpLinkRecipeXml);
    MpRecipeRegPar_Par.Enable := TRUE;
    MpRecipeRegPar_Par.PVName := ADR(AxisControl.Status.ProductSettingsName);
    MpRecipeRegPar_Par.Category := ADR(PARAMETERS_CATEGORY);
    MpRecipeRegPar_Par();
    ParametersPreview;
    ParametersEdit;

    AxisControl.Status.MachineSettingsName := AxisControl.Status.TaskName;
    brsstrcat(ADR(AxisControl.Status.MachineSettingsName), ADR(':MachineSettingsPreview'));
    MpRecipeRegPar_Cfg.MpLink := ADR(gMpLinkRecipeXml);
    MpRecipeRegPar_Cfg.Enable := TRUE;
    MpRecipeRegPar_Cfg.PVName := ADR(AxisControl.Status.MachineSettingsName);
    MpRecipeRegPar_Cfg.Category := ADR(MACHINE_CONFIGURATION_CATEGORY);
    MpRecipeRegPar_Cfg();
    MachineSettingsPreview;
    MachineSettingsEdit;

    // Activate RegPar FUBs
    WHILE NOT(MpRecipeRegPar_Par.Active OR MpRecipeRegPar_Par.Error) DO
        MpRecipeRegPar_Par();
    END_WHILE
    WHILE NOT(MpRecipeRegPar_Cfg.Active OR MpRecipeRegPar_Cfg.Error) DO
        MpRecipeRegPar_Cfg();
    END_WHILE

END_ACTION

ACTION RecipeCyclic:

	// HMI support handling
	IF (AxisRecipe.EditDialogOpened OR AxisRecipe.CreateDialogOpened) THEN
		IF (brsstrcmp(ADR(AxisRecipe.CategoryDropdown), ADR('Product')) = 0) THEN
			ParametersEdit := ParametersPreview;
		ELSIF (brsstrcmp(ADR(AxisRecipe.CategoryDropdown), ADR('Machine')) = 0) THEN
			MachineSettingsEdit := MachineSettingsPreview;
		END_IF
		AxisRecipe.EditDialogOpened := FALSE;
		AxisRecipe.CreateDialogOpened := FALSE;
	END_IF

	CASE AxisRecipe.State OF
		// Wait state
		REC_AXIS_WAIT:
			IF AxisRecipe.CreateRecipe THEN
				AxisRecipe.State := REC_AXIS_CREATE;
				AxisRecipe.CreateRecipe := FALSE;
			ELSIF AxisRecipe.SaveRecipe THEN
				AxisRecipe.State := REC_AXIS_SAVE;
				AxisRecipe.SaveRecipe := FALSE;
			ELSIF AxisRecipe.LoadRecipe THEN
				AxisRecipe.State := REC_AXIS_LOAD;
				AxisRecipe.LoadRecipe := FALSE;
			END_IF
		// Create recipe state
		REC_AXIS_CREATE:
			IF (brsstrcmp(ADR(AxisRecipe.CategoryDropdown), ADR('Product')) = 0) THEN
				ParametersPreview := ParametersEdit;
			ELSIF (brsstrcmp(ADR(AxisRecipe.CategoryDropdown), ADR('Machine')) = 0) THEN
				MachineSettingsPreview := MachineSettingsEdit;
			END_IF
			AxisRecipe.State := REC_AXIS_WAIT;
		// Load recipe state
		REC_AXIS_LOAD:
			IF (brsstrcmp(ADR(AxisRecipe.CategoryDropdown), ADR('Product')) = 0) THEN
				AxisControl.Parameters := ParametersPreview;
			ELSIF (brsstrcmp(ADR(AxisRecipe.CategoryDropdown), ADR('Machine')) = 0) THEN
				MachineSettings := MachineSettingsPreview;
			END_IF
			AxisRecipe.State := REC_AXIS_WAIT;
		// Save recipe state
		REC_AXIS_SAVE:
			IF (brsstrcmp(ADR(AxisRecipe.CategoryDropdown), ADR('Product')) = 0) THEN
				ParametersPreview := ParametersEdit;
			ELSIF (brsstrcmp(ADR(AxisRecipe.CategoryDropdown), ADR('Machine')) = 0) THEN
				MachineSettingsPreview := MachineSettingsEdit;
			END_IF
			AxisRecipe.State := REC_AXIS_WAIT;

	END_CASE;

	// Cyclic function block calls
	MpRecipeRegPar_Par.MpLink := ADR(gMpLinkRecipeXml);
	MpRecipeRegPar_Par();

	MpRecipeRegPar_Cfg.MpLink := ADR(gMpLinkRecipeXml);
	MpRecipeRegPar_Cfg();

END_ACTION
```

#### SimulationControl.st
```iecst
ACTION SimulationControl:

	// Automatic settings when project is in simulation
    IF NOT (DiagCpuIsARsim() OR DiagCpuIsSimulated()) THEN
        RETURN;
    END_IF

    IF ((MpAxisBasic_0.IsHomed = FALSE) AND (MpAxisBasic_0.Home = FALSE)) THEN
        AxisControl.Command.Reference := TRUE;
    END_IF

END_ACTION
```

### Program Logical/MachineControl/AxisTemplate/UnitTests/prototypeTest (ANSIC)

- AxisMgr.typ (reference to Logical/MachineControl/AxisTemplate/AxisMgr/AxisMgr.typ)

### Package Logical/MachineControl/AppAxis_1 - Package for mapp Axis Framework Application Axis

### Program Logical/MachineControl/AppAxis_1/AppAxis_1 (IEC) - Application axis manager

#### AxisMgr.typ - Local data types
```iecst
TYPE
	AxisSettingsType : {REDUND_UNREPLICABLE} 	STRUCT
		AxisFeatures : {REDUND_UNREPLICABLE} ARRAY[0..2]OF STRING[255];
		DriveConfiguration : {REDUND_UNREPLICABLE} McCfgPureVAxType;
		BaseConfiguration : {REDUND_UNREPLICABLE} McCfgAxType;
		BaseParam : {REDUND_UNREPLICABLE} McCfgAxMoveLimType;
	END_STRUCT;
	AxisMachineSettingsType : {REDUND_UNREPLICABLE} 	STRUCT
		ReferencePosition : {REDUND_UNREPLICABLE} LREAL := 0; (*[mm] Axis position after reference*)
	END_STRUCT;
	AxisControlCommandType : {REDUND_UNREPLICABLE} 	STRUCT
		UpdatePreviewParameters : {REDUND_UNREPLICABLE} BOOL;
		LoadRecipeParameters : {REDUND_UNREPLICABLE} BOOL;
		SaveRecipeParameters : {REDUND_UNREPLICABLE} BOOL;
		Power : {REDUND_UNREPLICABLE} BOOL;
		Reference : {REDUND_UNREPLICABLE} BOOL;
		MoveAbsolute : {REDUND_UNREPLICABLE} BOOL;
		MoveAdditive : {REDUND_UNREPLICABLE} BOOL;
		MoveToStart : {REDUND_UNREPLICABLE} BOOL;
		Abort : {REDUND_UNREPLICABLE} BOOL;
		Stop : {REDUND_UNREPLICABLE} BOOL;
		Reset : {REDUND_UNREPLICABLE} BOOL;
		JogPositive : {REDUND_UNREPLICABLE} BOOL;
		JogNegative : {REDUND_UNREPLICABLE} BOOL;
		Start : {REDUND_UNREPLICABLE} BOOL;
	END_STRUCT;
	AxisControlParametersType : {REDUND_UNREPLICABLE} 	STRUCT
		HomePosition : {REDUND_UNREPLICABLE} LREAL := 0;
		Position : {REDUND_UNREPLICABLE} LREAL := 0;
		Distance : {REDUND_UNREPLICABLE} LREAL := 180;
		Velocity : {REDUND_UNREPLICABLE} REAL := 360;
		Acceleration : {REDUND_UNREPLICABLE} REAL := 360;
		Deceleration : {REDUND_UNREPLICABLE} REAL := 360;
		JogVelocity : {REDUND_UNREPLICABLE} REAL := 100;
		StopDeceleration : {REDUND_UNREPLICABLE} REAL := 720; (*[mm/s2] Deceleration for stopping*)
		ProductNumber : {REDUND_UNREPLICABLE} INT := 0; (*Product Number*)
		ProductLength : {REDUND_UNREPLICABLE} REAL := 70; (*Real Product Length*)
	END_STRUCT;
	AxisControlStatusType : {REDUND_UNREPLICABLE} 	STRUCT
		TaskName : {REDUND_UNREPLICABLE} STRING[80];
		MachineSettingsName : {REDUND_UNREPLICABLE} STRING[255];
		ProductSettingsName : {REDUND_UNREPLICABLE} STRING[255];
		ProductPreviewSettingsName : {REDUND_UNREPLICABLE} STRING[255];
		Status : {REDUND_UNREPLICABLE} STRING[80]; (*Machine Status*)
		IsReady : {REDUND_UNREPLICABLE} BOOL;
		ErrorActive : {REDUND_UNREPLICABLE} BOOL;
		Busy : {REDUND_UNREPLICABLE} BOOL;
		ReferenceRequired : {REDUND_UNREPLICABLE} BOOL;
		Position : {REDUND_UNREPLICABLE} LREAL;
		Velocity : {REDUND_UNREPLICABLE} REAL;
		Current : {REDUND_UNREPLICABLE} REAL;
		LagError : {REDUND_UNREPLICABLE} LREAL;
		MotorTemperature : {REDUND_UNREPLICABLE} REAL;
		IsHomed : {REDUND_UNREPLICABLE} BOOL;
		IsPowered : {REDUND_UNREPLICABLE} BOOL;
	END_STRUCT;
	AxisControlType : {REDUND_UNREPLICABLE} 	STRUCT
		Command : {REDUND_UNREPLICABLE} AxisControlCommandType;
		Parameters : {REDUND_UNREPLICABLE} AxisControlParametersType;
		Status : {REDUND_UNREPLICABLE} AxisControlStatusType;
	END_STRUCT;
	StateEnum :
		(
		STATE_INIT,
		STATE_POWER_ON,
		STATE_HOME,
		STATE_REFERENCE,
		STATE_MOVE_TO_HOME_POSITION,
		STATE_READY,
		STATE_MANUAL_OPERATION,
		STATE_AUTOMATIC_OPERATION,
		STATE_STOPPING,
		STATE_STOPPED,
		STATE_ABORTING,
		STATE_ABORTED,
		STATE_CLEARING,
		STATE_RESETTING
		);
	ConfigurationStateEnum :
		(
		CONFIG_STATE_INIT,
		CONFIG_STATE_READ,
		CONFIG_STATE_WRITE,
		CONFIG_STATE_READY
		);
	ParameterStateEnum :
		(
		PAR_STATE_INIT,
		PAR_STATE_READ,
		PAR_STATE_WRITE,
		PAR_STATE_READY
		);
	AutomaticStateEnum :
		(
		AUTOMATIC_STATE_IDLE,
		AUTOMATIC_STATE_RUNNING
		);
	ManualStateEnum :
		(
		MANUAL_STATE_IDLE,
		MANUAL_STATE_JOG,
		MANUAL_STATE_MOVE,
		MANUAL_STATE_STOPPING
		);
	AxisRecipeType : 	STRUCT
		EditDialogOpened : BOOL;
		CreateDialogOpened : BOOL;
		SaveRecipe : BOOL;
		LoadRecipe : BOOL;
		CreateRecipe : BOOL;
		State : AxisRecipeStepEnum;
		CategoryDropdown : STRING[50];
	END_STRUCT;
	AxisRecipeStepEnum :
		(
		REC_AXIS_WAIT,
		REC_AXIS_LOAD,
		REC_AXIS_SAVE,
		REC_AXIS_CREATE,
		REC_AXIS_STORE_MACH_SETTINGS,
		REC_AXIS_FACTORY_RESET
		);
END_TYPE
```

- AxisMgr.var (reference to Logical/MachineControl/AxisTemplate/AxisMgr/AxisMgr.var)

#### SimulationControl.st - Simulation handling
```iecst
ACTION SimulationControl:
	// Automatic settings when project is in simulation
    IF NOT (DiagCpuIsARsim() OR DiagCpuIsSimulated()) THEN
        RETURN;
    END_IF

    IF ((MpAxisBasic_0.IsHomed = FALSE) AND (MpAxisBasic_0.Home = FALSE)) THEN
        AxisControl.Command.Reference := TRUE;
    END_IF

END_ACTION
```

#### AxisControlModes.st - Code that is specific to this axis
```iecst
ACTION AxisInit:

END_ACTION

ACTION AxisCyclic:

    MpAlarmXControl_SpeedNotSet.MpLink := ADR(gMpLinkAlarmXCoreAppAxis_1);
    MpAlarmXControl_SpeedNotSet.Enable := TRUE;
    MpAlarmXControl_SpeedNotSet.Name := ADR('AppAxis_1SpeedNotSet');
    MpAlarmXControl_SpeedNotSet();
    MpAlarmXControl_SpeedNotSet.Reset := FALSE;

END_ACTION

ACTION AxisManual:

    MpAxisParameters.Jog.Velocity := AxisControl.Parameters.JogVelocity;
    MpAxisParameters.Position := AxisControl.Parameters.Position;
    MpAxisParameters.Distance := AxisControl.Parameters.Distance;
    MpAxisParameters.Acceleration := AxisControl.Parameters.Acceleration;
    MpAxisParameters.Deceleration := AxisControl.Parameters.Deceleration;

    CASE ManualState OF
        MANUAL_STATE_IDLE:
            IF ((AxisControl.Command.JogNegative = TRUE) OR (AxisControl.Command.JogPositive = TRUE)) THEN
                ManualState := MANUAL_STATE_JOG;
            ELSIF ((AxisControl.Command.MoveAbsolute = TRUE) OR (AxisControl.Command.MoveAdditive = TRUE)) THEN
                MpAxisBasic_0.MoveAbsolute := AxisControl.Command.MoveAbsolute;
                MpAxisBasic_0.MoveAdditive := AxisControl.Command.MoveAdditive;
                AxisControl.Command.MoveAbsolute := FALSE;
                AxisControl.Command.MoveAdditive := FALSE;
                ManualState := MANUAL_STATE_MOVE;
            END_IF

        MANUAL_STATE_JOG:
            MpAxisBasic_0.JogNegative := AxisControl.Command.JogNegative;
            MpAxisBasic_0.JogPositive := AxisControl.Command.JogPositive;
            IF (AxisControl.Command.Stop = TRUE) THEN
                AxisControl.Command.Stop := FALSE;
                MpAxisBasic_0.Stop := TRUE;
                ManualState := MANUAL_STATE_STOPPING;
            ELSIF ((AxisControl.Command.JogNegative = FALSE) AND (AxisControl.Command.JogPositive = FALSE)) THEN
                MpAxisBasic_0.Stop := FALSE;
                MpAxisBasic_0.JogPositive := FALSE;
                MpAxisBasic_0.JogNegative := FALSE;
                ManualState := MANUAL_STATE_STOPPING;
            END_IF

        MANUAL_STATE_MOVE:
            IF (AxisControl.Command.Stop = TRUE) THEN
                MpAxisBasic_0.MoveAbsolute := FALSE;
                MpAxisBasic_0.MoveAdditive := FALSE;
                AxisControl.Command.Stop := FALSE;
                MpAxisBasic_0.Stop := TRUE;
                ManualState := MANUAL_STATE_STOPPING;
            ELSIF (InPositionEdgePos.Q = TRUE) THEN
                MpAxisBasic_0.MoveAbsolute := FALSE;
                MpAxisBasic_0.MoveAdditive := FALSE;
                ManualState := MANUAL_STATE_IDLE;
                State := STATE_READY;
            ELSIF ((AxisControl.Command.JogNegative = TRUE) OR (AxisControl.Command.JogPositive = TRUE)) THEN
                MpAxisBasic_0.MoveAbsolute := FALSE;
                MpAxisBasic_0.MoveAdditive := FALSE;
                ManualState := MANUAL_STATE_JOG;
            END_IF

        MANUAL_STATE_STOPPING:
            MpAxisBasic_0.JogNegative := FALSE;
            MpAxisBasic_0.JogPositive := FALSE;
            MpAxisBasic_0.MoveAbsolute := FALSE;
            MpAxisBasic_0.MoveAdditive := FALSE;

            IF (MpAxisBasic_0.MoveActive = FALSE) THEN
                ManualState := MANUAL_STATE_IDLE;
                State := STATE_READY;
            END_IF
    END_CASE

END_ACTION

ACTION AxisAutomatic:

    CASE AutomaticState OF
        AUTOMATIC_STATE_IDLE:
            IF (AxisControl.Command.Start = TRUE) THEN
                MpAlarmXControl_SpeedNotSet.Set := (MpAxisParameters.Velocity = 0);
                AxisControl.Command.Start := FALSE;
                AutomaticState := AUTOMATIC_STATE_RUNNING;
            END_IF

        AUTOMATIC_STATE_RUNNING:
            MpAxisBasic_0.MoveVelocity := TRUE;
            MpAxisParameters.Velocity := AxisControl.Parameters.Velocity;
            MpAxisParameters.Acceleration := AxisControl.Parameters.Acceleration;
            MpAxisParameters.Deceleration := AxisControl.Parameters.Deceleration;

            IF (AxisControl.Command.Stop = TRUE) THEN
                AxisControl.Command.Stop := FALSE;
                MpAxisBasic_0.MoveVelocity := FALSE;
                State := STATE_READY;
                AutomaticState := AUTOMATIC_STATE_IDLE;
            END_IF
    END_CASE

END_ACTION

ACTION AxisReset:

//    edge alarms don't require a reset
//    IF (MpAlarmXControl_SpeedNotSet.Set = TRUE) THEN
//        MpAlarmXControl_SpeedNotSet.Set := FALSE;
//        MpAlarmXControl_SpeedNotSet.ID := MpAlarmXControl_SpeedNotSet.InstanceID;
//        MpAlarmXControl_SpeedNotSet.Reset := TRUE;
//    END_IF

END_ACTION
```

- Recipe.st (reference to Logical/MachineControl/AxisTemplate/AxisMgr/Recipe.st)

#### LocalFunctions.fun - Functions for manual/automatic command
```iecst
{REDUND_ERROR} FUNCTION ManualCommand : BOOL (*Returns True if a manual command is active, false otherwise*) (*$GROUP=User,$CAT=User,$GROUPICON=User.png,$CATICON=User.png*)
	VAR_INPUT
		Commands : AxisControlCommandType;
	END_VAR
END_FUNCTION

{REDUND_ERROR} FUNCTION AutomaticCommand : BOOL (*Returns True if an automatic command is active*) (*$GROUP=User,$CAT=User,$GROUPICON=User.png,$CATICON=User.png*)
	VAR_INPUT
		Commands : AxisControlCommandType;
	END_VAR
END_FUNCTION
```

#### AutomaticCommand.st - Defines conditions for automatic mode
```iecst
// Returns True if an automatic command is active
FUNCTION AutomaticCommand

    AutomaticCommand := Commands.Start;

END_FUNCTION
```

#### AxisControl.typ - not listed in the package file held
```iecst
TYPE
	AxisSettingsType : {REDUND_UNREPLICABLE} 	STRUCT
		AxisFeatures : {REDUND_UNREPLICABLE} ARRAY[0..2]OF STRING[255];
		DriveConfiguration : {REDUND_UNREPLICABLE} McCfgPureVAxType;
		BaseConfiguration : {REDUND_UNREPLICABLE} McCfgAxType;
		MechanicalParameter : {REDUND_UNREPLICABLE} McCfgAcpMechElmType;
		ControllerParameter : {REDUND_UNREPLICABLE} McCfgAcpCtrlType;
	END_STRUCT;
	AxisMachineSettingsType : {REDUND_UNREPLICABLE} 	STRUCT
		ReferencePosition : {REDUND_UNREPLICABLE} LREAL := 0; (*[mm] Axis position after reference*)
	END_STRUCT;
	AxisControlCommandType : {REDUND_UNREPLICABLE} 	STRUCT
		UpdatePreviewParameters : {REDUND_UNREPLICABLE} BOOL;
		LoadRecipeParameters : {REDUND_UNREPLICABLE} BOOL;
		SaveRecipeParameters : {REDUND_UNREPLICABLE} BOOL;
		Power : {REDUND_UNREPLICABLE} BOOL;
		Reference : {REDUND_UNREPLICABLE} BOOL;
		MoveAbsolute : {REDUND_UNREPLICABLE} BOOL;
		MoveAdditive : {REDUND_UNREPLICABLE} BOOL;
		MoveToStart : {REDUND_UNREPLICABLE} BOOL;
		Abort : {REDUND_UNREPLICABLE} BOOL;
		Stop : {REDUND_UNREPLICABLE} BOOL;
		Reset : {REDUND_UNREPLICABLE} BOOL;
		JogPositive : {REDUND_UNREPLICABLE} BOOL;
		JogNegative : {REDUND_UNREPLICABLE} BOOL;
		Start : {REDUND_UNREPLICABLE} BOOL;
	END_STRUCT;
	AxisControlParametersType : {REDUND_UNREPLICABLE} 	STRUCT
		HomePosition : {REDUND_UNREPLICABLE} LREAL := 0;
		Position : {REDUND_UNREPLICABLE} LREAL := 0;
		Distance : {REDUND_UNREPLICABLE} LREAL := 180;
		Velocity : {REDUND_UNREPLICABLE} REAL := 360;
		Acceleration : {REDUND_UNREPLICABLE} REAL := 360;
		Deceleration : {REDUND_UNREPLICABLE} REAL := 360;
		JogVelocity : {REDUND_UNREPLICABLE} REAL := 100;
		StopDeceleration : {REDUND_UNREPLICABLE} REAL := 720; (*[mm/s2] Deceleration for stopping*)
		ProductNumber : {REDUND_UNREPLICABLE} INT := 0; (*Product Number*)
		ProductLength : {REDUND_UNREPLICABLE} REAL := 70; (*Real Product Length*)
	END_STRUCT;
	AxisControlStatusType : {REDUND_UNREPLICABLE} 	STRUCT
		TaskName : {REDUND_UNREPLICABLE} STRING[80];
		MachineSettingsName : {REDUND_UNREPLICABLE} STRING[255];
		ProductSettingsName : {REDUND_UNREPLICABLE} STRING[255];
		ProductPreviewSettingsName : {REDUND_UNREPLICABLE} STRING[255];
		Status : {REDUND_UNREPLICABLE} STRING[80]; (*Machine Status*)
		IsReady : {REDUND_UNREPLICABLE} BOOL;
		ErrorActive : {REDUND_UNREPLICABLE} BOOL;
		Busy : {REDUND_UNREPLICABLE} BOOL;
		ReferenceRequired : {REDUND_UNREPLICABLE} BOOL;
		Position : {REDUND_UNREPLICABLE} LREAL;
		Velocity : {REDUND_UNREPLICABLE} REAL;
		Current : {REDUND_UNREPLICABLE} REAL;
		LagError : {REDUND_UNREPLICABLE} LREAL;
		MotorTemperature : {REDUND_UNREPLICABLE} REAL;
		IsHomed : {REDUND_UNREPLICABLE} BOOL;
		IsPowered : {REDUND_UNREPLICABLE} BOOL;
	END_STRUCT;
	AxisControlType : {REDUND_UNREPLICABLE} 	STRUCT
		Command : {REDUND_UNREPLICABLE} AxisControlCommandType;
		Parameters : {REDUND_UNREPLICABLE} AxisControlParametersType;
		Status : {REDUND_UNREPLICABLE} AxisControlStatusType;
	END_STRUCT;
	StateEnum :
		(
		STATE_INIT,
		STATE_POWER_ON,
		STATE_HOME,
		STATE_REFERENCE,
		STATE_MOVE_TO_HOME_POSITION,
		STATE_READY,
		STATE_MANUAL_OPERATION,
		STATE_AUTOMATIC_OPERATION,
		STATE_STOPPING,
		STATE_STOPPED,
		STATE_ABORTING,
		STATE_ABORTED,
		STATE_CLEARING,
		STATE_RESETTING
		);
	ConfigurationStateEnum :
		(
		CONFIG_STATE_INIT,
		CONFIG_STATE_READ,
		CONFIG_STATE_WRITE,
		CONFIG_STATE_READY
		);
	ParameterStateEnum :
		(
		PAR_STATE_INIT,
		PAR_STATE_READ,
		PAR_STATE_WRITE,
		PAR_STATE_READY
		);
	AutomaticStateEnum :
		(
		AUTOMATIC_STATE_IDLE,
		AUTOMATIC_STATE_RUNNING
		);
	ManualStateEnum :
		(
		MANUAL_STATE_IDLE,
		MANUAL_STATE_JOG,
		MANUAL_STATE_MOVE,
		MANUAL_STATE_STOPPING
		);
	AxisRecipeType : 	STRUCT
		EditDialogOpened : BOOL;
		CreateDialogOpened : BOOL;
		SaveRecipe : BOOL;
		LoadRecipe : BOOL;
		CreateRecipe : BOOL;
		State : AxisRecipeStepEnum;
		CategoryDropdown : STRING[50];
	END_STRUCT;
	AxisRecipeStepEnum :
		(
		REC_AXIS_WAIT,
		REC_AXIS_LOAD,
		REC_AXIS_SAVE,
		REC_AXIS_CREATE,
		REC_AXIS_STORE_MACH_SETTINGS,
		REC_AXIS_FACTORY_RESET
		);
END_TYPE
```

#### AxisControl.st - not listed in the package file held
```iecst
//***********************************************************************************************************************
//* Copyright: B&R Industrial Automation GmbH
//* Description: This program implements an axis control
//***********************************************************************************************************************

PROGRAM _INIT

    ST_name(0, ADR(AxisControl.Status.TaskName), 0);

	RecipeInit;
	ConfigurationInit;
	ParameterInit;

	// Inititialize mapp function blocks
    MpAlarmXCore_0.Enable := TRUE;
	MpAxisBasic_0.Enable := TRUE;

	AxisInit;
END_PROGRAM

PROGRAM _CYCLIC

    MpAxisBasic_0.MpLink := ADR(gMpLinkAppAxis_1);
    MC_BR_CheckRestorePositionData_0.Axis := ADR(gMpLinkAppAxis_1);

	// Call all actions
    SimulationControl;
    AxisStateMachine;
    AxisCyclic;
    RecipeCyclic;

	// Assign MpLink
	MpAlarmXCore_0.MpLink := ADR(gMpLinkAlarmXCoreAppAxis_1);

	// Call function block
    MpAlarmXCore_0();

END_PROGRAM

PROGRAM _EXIT

	// Disable the function blocls to unlink the MpLinks.
	// Do NOT disable MpAxisBasic, as this can cause problems during project transfer.
    MpRecipeRegPar_Par.Enable := FALSE;
	MpRecipeRegPar_Cfg.Enable := FALSE;
	MpAlarmXCore_0.Enable := FALSE;

	// Call function blocks
	MpRecipeRegPar_Par();
	MpRecipeRegPar_Cfg();
	MpAlarmXCore_0();

END_PROGRAM
```

### Package Logical/MachineControl/AppAxis_1/UnitTests - Multiple variants of valid test sets

### Program Logical/MachineControl/AppAxis_1/UnitTests/ConvTest

#### Set_SetupTeardown.c
```c
/********************************************************************
 * COPYRIGHT --
 ********************************************************************
 * Program: -
 * Author:
 * Created:
 ********************************************************************
 * Tests for ...
 ********************************************************************/

#include <bur/plctypes.h>

#ifdef _DEFAULT_INCLUDES
#include <AsDefault.h>
#endif

#include <stdbool.h>
#include "UnitTest.h"

_SETUP_SET(void)
{
    // wait until the axis is ready
    TEST_BUSY_CONDITION(AxisControl.Status.IsReady == false);

    TEST_DONE;
}

_TEARDOWN_SET(void)
{
	TEST_DONE;
}

_SETUP_TEST(void)
{
    testState = TEST_STATE_ARRANGE;
	TEST_DONE;
}

_TEARDOWN_TEST(void)
{
    AxisControl.Command.JogNegative = false;
    AxisControl.Command.JogPositive = false;
    AxisControl.Command.MoveToStart = false;
    AxisControl.Command.Start = false;
    TEST_BUSY_CONDITION(AxisControl.Status.Velocity > 0.001);
    TEST_BUSY_CONDITION(AxisControl.Status.Velocity < -0.001);

	TEST_DONE;
}

_TEST powerOnTest(void)
{
    switch (testState)
    {
        case TEST_STATE_ARRANGE:
            // Arrange
            AxisControl.Command.Power = true;
            TEST_BUSY_CONDITION(AxisControl.Status.Busy == false);
            testState = TEST_STATE_ACT;
            break;

        case TEST_STATE_ACT:
            // Act
            TEST_BUSY_CONDITION(AxisControl.Status.Busy);
            testState = TEST_STATE_ASSERT;
            break;

        case TEST_STATE_ASSERT:
            // Assert
            TEST_ASSERT(AxisControl.Status.IsPowered);
            testState = TEST_STATE_DONE;
            break;

        case TEST_STATE_DONE:
            /* test is done */
            TEST_DONE;
    }

    TEST_BUSY;
}

_TEST homeTest(void)
{
    switch (testState)
    {
        case TEST_STATE_ARRANGE:
            // Arrange
            AxisControl.Command.Home = true;
            TEST_BUSY_CONDITION(AxisControl.Status.Busy == false);
            testState = TEST_STATE_ACT;
            break;

        case TEST_STATE_ACT:
            // Act
            TEST_BUSY_CONDITION(AxisControl.Status.Busy);
            testState = TEST_STATE_ASSERT;
            break;

        case TEST_STATE_ASSERT:
            // Assert
            TEST_ASSERT(AxisControl.Status.IsHomed);
            testState = TEST_STATE_DONE;
            break;

        case TEST_STATE_DONE:
            /* test is done */
            TEST_DONE;
    }

    TEST_BUSY;
}

_TEST jogNegativeTest(void)
{
    switch (testState)
    {
        case TEST_STATE_ARRANGE:
            // Arrange
            AxisControl.Parameters.JogVelocity = 5.0;
            testState = TEST_STATE_ACT;
            break;

        case TEST_STATE_ACT:
            // Act
            AxisControl.Command.JogNegative = true;
            TEST_BUSY_CONDITION(AxisControl.Status.Velocity > -0.01);
            testState = TEST_STATE_ASSERT;
            break;

        case TEST_STATE_ASSERT:
            // Assert
            TEST_ASSERT_REAL_WITHIN(0.01, -5.0, AxisControl.Status.Velocity);
            AxisControl.Command.JogNegative = false;
            testState = TEST_STATE_DONE;
            break;

        case TEST_STATE_DONE:
            /* test is done */
            TEST_DONE;
    }

    TEST_BUSY;
}

_TEST jogPositiveTest(void)
{
    switch (testState)
    {
        case TEST_STATE_ARRANGE:
            // Arrange
            AxisControl.Parameters.JogVelocity = 6.0;
            testState = TEST_STATE_ACT;
            break;

        case TEST_STATE_ACT:
            // Act
            AxisControl.Command.JogPositive = true;
            TEST_BUSY_CONDITION(AxisControl.Status.Velocity < 0.01);
            testState = TEST_STATE_ASSERT;
            break;

        case TEST_STATE_ASSERT:
            // Assert
            TEST_ASSERT_REAL_WITHIN(0.01, 6.0, AxisControl.Status.Velocity);
            AxisControl.Command.JogPositive = false;
            testState = TEST_STATE_DONE;
            break;

        case TEST_STATE_DONE:
            /* test is done */
            TEST_DONE;
    }

    TEST_BUSY;
}

/*
B+R UnitTest: This is generated code.
Do not edit! Do not move!
Description: UnitTest Testprogramm infrastructure (TestSet).
LastUpdated: 2021-09-29 12:12:33Z
By B+R UnitTest Helper Version: 2.0.1.59
*/
UNITTEST_FIXTURES(fixtures)
{
	new_TestFixture("powerOnTest", powerOnTest),
	new_TestFixture("homeTest", homeTest),
	new_TestFixture("jogNegativeTest", jogNegativeTest),
	new_TestFixture("jogPositiveTest", jogPositiveTest),
};

UNITTEST_CALLER_COMPLETE_EXPLICIT(Set_SetupTeardown, "Set_SetupTeardown", setupTest, teardownTest, fixtures, setupSet, teardownSet, 0);
```

### Program Logical/MachineControl/CrossCutter/CrossCutter (IEC)

#### AxisControl.st - Init, cyclic, exit code
```iecst
//***********************************************************************************************************************
//* Copyright: B&R Industrial Automation GmbH
//* Description: This program implements an axis control
//**********************************************************************************************************************

PROGRAM _INIT

    ST_name(0, ADR(AxisControl.Status.TaskName), 0);
    RecipeInit;

    MpAlarmXCore_0.Enable := TRUE;
    ConfigurationInit;

    MpAxisBasic_0.Enable := TRUE;

    AxisInit;
END_PROGRAM

PROGRAM _CYCLIC

    MpAxisBasic_0.MpLink := ADR(gAxisCrossCutter);
    MC_BR_CheckRestorePositionData_0.Axis := ADR(gAxisCrossCutter);

    SimulationControl;
    AxisStateMachine;
    AxisCyclic;
    RecipeCyclic;

    MpAlarmXCore_0.MpLink := ADR(gAlarmXCore_Cutter);
    MpAlarmXCore_0();

END_PROGRAM

PROGRAM _EXIT

    MpRecipeRegPar_MachineFB.Enable := FALSE;
    MpRecipeRegPar_MachineFB();

    MpRecipeRegPar_UserFB.Enable := FALSE;
    MpRecipeRegPar_UserFB();

    MpRecipeRegPar_PreFB.Enable := FALSE;
    MpRecipeRegPar_PreFB();

    MpRecipeRegPar_UserPreFB.Enable := FALSE;
    MpRecipeRegPar_UserPreFB();

    MpAxisBasic_0.Enable := FALSE;
    MpAxisBasic_0();

    MC_BR_CamAutomatCommandFB.Enable := FALSE;
    MC_BR_CamAutomatCommandFB();

    MpAlarmXCore_0.Enable := FALSE;
    MpAlarmXCore_0();

END_PROGRAM
```

#### SimulationControl.st
```iecst
ACTION SimulationControl:

	IF NOT (DiagCpuIsARsim() OR DiagCpuIsSimulated()) THEN
		RETURN;
	END_IF

    IF ((MpAxisBasic_0.IsHomed = FALSE) AND (MpAxisBasic_0.Home = FALSE)) THEN
        AxisControl.Command.Reference := TRUE;
    END_IF

END_ACTION
```

#### AxisControlModes.st
```iecst
ACTION AxisInit:

    MC_BR_CamAutomatCommandFB.Enable := TRUE;

    MC_BR_CamAutomatGetParFB.Command := mcGET_PAR_ACTUAL;
    MC_BR_CamAutomatGetParFB.Execute := TRUE;

    MC_BR_CamAutomatSetParFB.Command := mcSET_UPDATE_FROM_ADR;
    MC_BR_CamAutomatSetParFB.AdvancedParameters.ParLock := mcCAMAUT_UNLOCK_SYNCHRON;

    MpRegMarkDetectionFB.Enable := TRUE;
    MpRegMarkDetectionConfigFB.Enable := TRUE;
    MpRegMarkDetectionConfigFB.MpLink := ADR(gRegMarkDetection_Cutter);
    MpRegMarkDetectionConfigFB.Configuration := ADR(RegistrationControl.Configuration);
    WHILE NOT MpRegMarkDetectionConfigFB.Active AND NOT MpRegMarkDetectionConfigFB.Error DO
        MpRegMarkDetectionConfigFB();
    END_WHILE
    MpRegMarkDetectionConfigFB.Load := TRUE;
    MpRegMarkDetectionConfigFB();

    MC_BR_PhasingFB.Velocity := 90;
    MC_BR_PhasingFB.Acceleration := 90;
    MC_BR_PhasingFB.AdvancedParameters.ShiftMode := mcSHIFT_RELATIVE;

    END_ACTION

ACTION AxisCyclic:

    IF ((MpRegMarkDetectionConfigFB.Active = TRUE) AND (state = STATE_INIT)) THEN
        MpRegMarkDetectionConfigFB.Load := TRUE;
    END_IF

    IF (MpRecipeRegPar_UserFB.UpdateNotification) THEN
        UpdateCamAutomat;
        UpdateRegistrationControl;
    END_IF

    MC_BR_CamAutomatGetParFB.CamAutomat.DataAddress := ADR(McCamAutPar);
    MC_BR_CamAutomatGetParFB.Slave := ADR(gAxisCrossCutter);
    MC_BR_CamAutomatGetParFB();
    IF (MC_BR_CamAutomatGetParFB.Done = TRUE) THEN
        MC_BR_CamAutomatGetParFB.Execute := FALSE;
    END_IF
    i:=i + 1;

    MC_BR_CamAutomatSetParFB.Slave := ADR(gAxisCrossCutter);
    MC_BR_CamAutomatSetParFB.CamAutomat.DataAddress := ADR(McCamAutPar);
    MC_BR_CamAutomatSetParFB();
    IF (MC_BR_CamAutomatSetParFB.Done = TRUE) THEN
        MC_BR_CamAutomatSetParFB.Execute := FALSE;
    END_IF

    MC_BR_CamAutomatCommandFB.Slave := ADR(gAxisCrossCutter);
    MC_BR_CamAutomatCommandFB();

    MpRegMarkDetectionFB.MpLink := ADR(gRegMarkDetection_Cutter);
    MpRegMarkDetectionFB();

    MpRegMarkDetectionConfigFB.MpLink := ADR(gRegMarkDetection_Cutter);
    MpRegMarkDetectionConfigFB.Configuration := ADR(RegistrationControl.Configuration);
    MpRegMarkDetectionConfigFB();
    IF (MpRegMarkDetectionConfigFB.CommandDone = TRUE) THEN
        MpRegMarkDetectionConfigFB.Load := FALSE;
        MpRegMarkDetectionConfigFB.Save := FALSE;
    END_IF

    MC_BR_PhasingFB.Slave := ADR(gAxisCrossCutter);
    MC_BR_PhasingFB();

    IF (state <> STATE_AUTOMATIC_OPERATION) THEN
        AutomaticState := 0;
    END_IF

    MpAlarmXControlProductLengthFB.MpLink := ADR(gAlarmXCore_Cutter);
    MpAlarmXControlProductLengthFB.Enable := TRUE;
    MpAlarmXControlProductLengthFB.Name := ADR('CutterInvalidProductLength');
    MpAlarmXControlProductLengthFB();
    MpAlarmXControlProductLengthFB.Reset := FALSE;

    END_ACTION

ACTION UpdateCamAutomat:

    McCamAutPar.Common.Master.MasterStartInterval := AxisControl.Parameters.ProductLength;

    McCamAutPar.State[1].MasterFactor := LREAL_TO_DINT(AxisControl.Parameters.SyncAngle);
    McCamAutPar.State[1].SlaveFactor := LREAL_TO_DINT(AxisControl.Parameters.SyncAngle);
    McCamAutPar.State[1].CompensationParameters.MasterCompDistance := AxisControl.Parameters.DistanceFromSensorToCut;

    McCamAutPar.State[2].MasterFactor := LREAL_TO_DINT(AxisControl.Parameters.SyncAngle);
    McCamAutPar.State[2].SlaveFactor := LREAL_TO_DINT(AxisControl.Parameters.SyncAngle);
    McCamAutPar.State[2].CompensationParameters.MasterCompDistance := AxisControl.Parameters.ProductLength;
    McCamAutPar.State[2].CompensationParameters.SlaveCompDistance := 360.0 /  AxisControl.Parameters.NumberOfKnives;

    McCamAutPar.State[3].CompensationParameters.MasterCompDistance := AxisControl.Parameters.ProductLength;
    CASE  AxisControl.Parameters.NumberOfKnives OF
        1:
            McCamAutPar.State[3].CompensationParameters.SlaveCompDistance := 270.0;
        2:
            McCamAutPar.State[3].CompensationParameters.SlaveCompDistance := 90.0;
    END_CASE

    IF ((MpAxisBasic_0.Active = TRUE) AND (MC_BR_CamAutomatCommandFB.Running = FALSE)) THEN
        MC_BR_CamAutomatSetParFB.Execute := TRUE;
    END_IF

    END_ACTION

ACTION UpdateRegistrationControl:

    RegistrationControl.Configuration.Measurement.Product.Length.Value := AxisControl.Parameters.ProductLength;
    RegistrationControl.Configuration.Measurement.Interval.Length.Value := AxisControl.Parameters.ProductLength;
    RegistrationControl.Configuration.Detection.MarkWidthMonitoring.MaximumWidth := AxisControl.Parameters.MaxPrintMarkLength;
    RegistrationControl.Configuration.Detection.MarkWidthMonitoring.MinimumWidth := AxisControl.Parameters.MinPrintMarkLength;

    MpRegMarkDetectionConfigFB.Save := TRUE;

    END_ACTION

ACTION AxisManual:

    MpAxisParameters.Jog.Velocity := AxisControl.Parameters.JogVelocity;
    MpAxisParameters.Position := AxisControl.Parameters.Position;
    MpAxisParameters.Distance := AxisControl.Parameters.Distance;
    MpAxisParameters.Acceleration := AxisControl.Parameters.Acceleration;
    MpAxisParameters.Deceleration := AxisControl.Parameters.Deceleration;

    CASE ManualState OF
        MANUAL_STATE_IDLE:
            IF ((AxisControl.Command.JogNegative = TRUE) OR (AxisControl.Command.JogPositive = TRUE)) THEN
                ManualState := MANUAL_STATE_JOG;
            ELSIF ((AxisControl.Command.MoveAbsolute = TRUE) OR (AxisControl.Command.MoveAdditive = TRUE)) THEN
                MpAxisBasic_0.MoveAbsolute := AxisControl.Command.MoveAbsolute;
                MpAxisBasic_0.MoveAdditive := AxisControl.Command.MoveAdditive;
                AxisControl.Command.MoveAbsolute := FALSE;
                AxisControl.Command.MoveAdditive := FALSE;
                ManualState := MANUAL_STATE_MOVE;
            END_IF

        MANUAL_STATE_JOG:
            MpAxisBasic_0.JogNegative := AxisControl.Command.JogNegative;
            MpAxisBasic_0.JogPositive := AxisControl.Command.JogPositive;
            IF (AxisControl.Command.Stop = TRUE) THEN
                AxisControl.Command.Stop := FALSE;
                MpAxisBasic_0.Stop := TRUE;
                ManualState := MANUAL_STATE_STOPPING;
            ELSIF ((AxisControl.Command.JogNegative = FALSE) AND (AxisControl.Command.JogPositive = FALSE)) THEN
                MpAxisBasic_0.Stop := FALSE;
                MpAxisBasic_0.JogPositive := FALSE;
                MpAxisBasic_0.JogNegative := FALSE;
                ManualState := MANUAL_STATE_STOPPING;
            END_IF

        MANUAL_STATE_MOVE:
            IF (AxisControl.Command.Stop = TRUE) THEN
                MpAxisBasic_0.MoveAbsolute := FALSE;
                MpAxisBasic_0.MoveAdditive := FALSE;
                AxisControl.Command.Stop := FALSE;
                MpAxisBasic_0.Stop := TRUE;
                ManualState := MANUAL_STATE_STOPPING;
            ELSIF (InPositionEdgePos.Q = TRUE) THEN
                MpAxisBasic_0.MoveAbsolute := FALSE;
                MpAxisBasic_0.MoveAdditive := FALSE;
                ManualState := MANUAL_STATE_IDLE;
                state := STATE_READY;
            ELSIF ((AxisControl.Command.JogNegative = TRUE) OR (AxisControl.Command.JogPositive = TRUE)) THEN
                MpAxisBasic_0.MoveAbsolute := FALSE;
                MpAxisBasic_0.MoveAdditive := FALSE;
                ManualState := MANUAL_STATE_JOG;
            END_IF

        MANUAL_STATE_STOPPING:
            MpAxisBasic_0.JogNegative := FALSE;
            MpAxisBasic_0.JogPositive := FALSE;
            MpAxisBasic_0.MoveAbsolute := FALSE;
            MpAxisBasic_0.MoveAdditive := FALSE;

            IF (MpAxisBasic_0.MoveActive = FALSE) THEN
                ManualState := MANUAL_STATE_IDLE;
                state := STATE_READY;
            END_IF
    END_CASE

    END_ACTION

ACTION AxisAutomatic:

    MpAlarmXControlProductLengthFB.Set := (AxisControl.Parameters.ProductLength = 0);

    MpAxisParameters.Velocity := AxisControl.Parameters.Velocity;
    MpAxisParameters.Acceleration := AxisControl.Parameters.Acceleration;
    MpAxisParameters.Deceleration := AxisControl.Parameters.Deceleration;

    MC_BR_CamAutomatCommandFB.SetSignal1 := FALSE;
    CASE AutomaticState OF
        0:
            MpRegMarkDetectionFB.Detect := TRUE;
            MpRegMarkDetectionFB.Search := TRUE;
            IF (MpRegMarkDetectionFB.SearchDone = TRUE) THEN
                MC_BR_PhasingFB.Enable := TRUE;
                AutomaticState := 1;
                MpRegMarkDetectionFB.Search := FALSE;
            END_IF

        1:
            IF (MpRegMarkDetectionFB.Info.Detection.TotalValidMarks <> RegistrationControl.LastValidMarks) THEN
                RegistrationControl.LastValidMarks := MpRegMarkDetectionFB.Info.Detection.TotalValidMarks;
                IF (RegistrationControl.ActualProductLength > 60) THEN
                    RegistrationControl.PhaseShift := AxisControl.Parameters.ProductLength - RegistrationControl.ActualProductLength;
                END_IF

                IF (MC_BR_CamAutomatCommandFB.Running = FALSE) THEN
                    MC_BR_CamAutomatCommandFB.SetSignal1 := FALSE;
                    MC_BR_CamAutomatCommandFB.ResetSignal1 := TRUE;
                    MC_BR_CamAutomatCommandFB.Start := (MC_BR_CamAutomatCommandFB.Start = FALSE);
                ELSIF (MC_BR_CamAutomatCommandFB.ActualStateIndex > 0) THEN
                    MC_BR_CamAutomatCommandFB.ResetSignal1 := FALSE;
                    MC_BR_CamAutomatCommandFB.SetSignal1 := TRUE;
                END_IF
            END_IF

            IF ((MC_BR_PhasingFB.PhaseShift <> RegistrationControl.PhaseShift) AND (MC_BR_CamAutomatCommandFB.ActualStateIndex > 0)) THEN
                MC_BR_PhasingFB.PhaseShift := RegistrationControl.PhaseShift;
                MC_BR_PhasingFB.StartShift := TRUE;
            END_IF

            IF EDGEPOS(MC_BR_PhasingFB.ShiftAttained = TRUE) THEN
                MC_BR_PhasingFB.StartShift := FALSE;
            END_IF

            IF (AxisControl.Command.Stop = TRUE) THEN
                AxisControl.Command.Stop := FALSE;
                MC_BR_PhasingFB.Enable := FALSE;
                MC_BR_CamAutomatCommandFB.SetSignal2 := TRUE;
                AutomaticState := 10;
            END_IF

        10:
            IF (MC_BR_CamAutomatCommandFB.Running = FALSE) THEN
                state := STATE_READY;
            END_IF

    END_CASE

    AxisControl.Status.ActualProductLength := RegistrationControl.ActualProductLength;
    AxisControl.Status.ValidProducts := MpRegMarkDetectionFB.Info.Detection.TotalValidMarks;

    END_ACTION

ACTION AxisReset:

    //    edge alarms don't require a reset
    //    IF (MpAlarmXControlProductLengthFB.Set = TRUE) THEN
    //        MpAlarmXControlProductLengthFB.Set := FALSE;
    //        MpAlarmXControlProductLengthFB.ID := MpAlarmXControlProductLengthZeroFB.InstanceID;
    //        MpAlarmXControlProductLengthFB.Reset := TRUE;
    //    END_IF

    END_ACTION
```

#### ManualCommand.st
```iecst
(* Returns True if a manual command is active, false otherwise *)
FUNCTION ManualCommand
    ManualCommand := Commands.JogNegative OR Commands.JogPositive OR Commands.MoveAbsolute OR Commands.MoveAdditive;
END_FUNCTION
```

#### AutomaticCommand.st
```iecst
(* Returns True if an automatic command is active
FUNCTION AutomaticCommand

    AutomaticCommand := Commands.Start;

END_FUNCTION
```

#### Types.typ - not listed in the package file held
```iecst
TYPE
	AxisMachineSettingsType : {REDUND_UNREPLICABLE} 	STRUCT
		ReferencePosition : {REDUND_UNREPLICABLE} LREAL := 0.0; (*[deg] Position when the axis is referenced*)
		AxisFeatures : {REDUND_UNREPLICABLE} ARRAY[0..2]OF STRING[255] := ['CamAut_cutting',''];
		DriveConfiguration : {REDUND_UNREPLICABLE} McCfgPureVAxType := (0);
		BaseConfiguration : {REDUND_UNREPLICABLE} McCfgAxType;
	END_STRUCT;
	AxisControlCommandType : {REDUND_UNREPLICABLE} 	STRUCT
		UpdatePreviewParameters : {REDUND_UNREPLICABLE} BOOL;
		ResetEditParameters : {REDUND_UNREPLICABLE} BOOL;
		Power : {REDUND_UNREPLICABLE} BOOL;
		Reference : {REDUND_UNREPLICABLE} BOOL;
		MoveToStart : {REDUND_UNREPLICABLE} BOOL;
		MoveAbsolute : {REDUND_UNREPLICABLE} BOOL;
		MoveAdditive : {REDUND_UNREPLICABLE} BOOL;
		Abort : {REDUND_UNREPLICABLE} BOOL;
		Stop : {REDUND_UNREPLICABLE} BOOL;
		Reset : {REDUND_UNREPLICABLE} BOOL;
		JogPositive : {REDUND_UNREPLICABLE} BOOL;
		JogNegative : {REDUND_UNREPLICABLE} BOOL;
		Start : {REDUND_UNREPLICABLE} BOOL;
	END_STRUCT;
	AxisControlParametersType : {REDUND_UNREPLICABLE} 	STRUCT
		HomePosition : {REDUND_UNREPLICABLE} LREAL := 0;
		Position : {REDUND_UNREPLICABLE} LREAL := 0;
		Distance : {REDUND_UNREPLICABLE} LREAL := 180;
		Velocity : {REDUND_UNREPLICABLE} REAL := 360;
		Acceleration : {REDUND_UNREPLICABLE} REAL := 360;
		Deceleration : {REDUND_UNREPLICABLE} REAL := 360;
		JogVelocity : {REDUND_UNREPLICABLE} REAL := 360;
		StopDeceleration : {REDUND_UNREPLICABLE} REAL := 720; (*[mm/s2] Deceleration for stopping*)
		SyncAngle : {REDUND_UNREPLICABLE} LREAL := 45; (*Product Number*)
		DistanceFromSensorToCut : {REDUND_UNREPLICABLE} LREAL := 100; (*Real Product Length*)
		NumberOfKnives : {REDUND_UNREPLICABLE} USINT := 2;
		ProductLength : {REDUND_UNREPLICABLE} LREAL := 70;
		MinPrintMarkLength : {REDUND_UNREPLICABLE} LREAL := 7; (*[mm] Minimum product length, used for product detection*)
		MaxPrintMarkLength : {REDUND_UNREPLICABLE} LREAL := 15; (*[mm] Minimum print mark length, used for product detection*)
	END_STRUCT;
	AxisControlStatusType : {REDUND_UNREPLICABLE} 	STRUCT
		TaskName : {REDUND_UNREPLICABLE} STRING[80];
		MachineSettingsName : {REDUND_UNREPLICABLE} STRING[255];
		ProductSettingsName : {REDUND_UNREPLICABLE} STRING[255];
		ProductPreviewSettingsName : {REDUND_UNREPLICABLE} STRING[255];
		Status : {REDUND_UNREPLICABLE} STRING[80]; (*Machine Status*)
		IsReady : {REDUND_UNREPLICABLE} BOOL;
		ErrorActive : {REDUND_UNREPLICABLE} BOOL;
		Busy : {REDUND_UNREPLICABLE} BOOL;
		ReferenceRequired : {REDUND_UNREPLICABLE} BOOL;
		Position : {REDUND_UNREPLICABLE} LREAL;
		Velocity : {REDUND_UNREPLICABLE} REAL;
		Current : {REDUND_UNREPLICABLE} REAL;
		LagError : {REDUND_UNREPLICABLE} LREAL;
		MotorTemperature : {REDUND_UNREPLICABLE} REAL;
		IsHomed : {REDUND_UNREPLICABLE} BOOL;
		IsPowered : {REDUND_UNREPLICABLE} BOOL;
		ActualProductLength : {REDUND_UNREPLICABLE} LREAL;
		ValidProducts : {REDUND_UNREPLICABLE} UDINT;
	END_STRUCT;
	AxisControlType : {REDUND_UNREPLICABLE} 	STRUCT
		Command : {REDUND_UNREPLICABLE} AxisControlCommandType;
		Parameters : {REDUND_UNREPLICABLE} AxisControlParametersType;
		Status : {REDUND_UNREPLICABLE} AxisControlStatusType;
	END_STRUCT;
	stateEnum :
		(
		STATE_INIT,
		STATE_POWER_ON,
		STATE_HOME,
		STATE_REFERENCE,
		STATE_MOVE_TO_HOME_POSITION,
		STATE_READY,
		STATE_MANUAL_OPERATION,
		STATE_AUTOMATIC_OPERATION,
		STATE_STOPPING,
		STATE_STOPPED,
		STATE_ABORTING,
		STATE_ABORTED,
		STATE_CLEARING,
		STATE_RESETTING
		);
	configurationStateEnum :
		(
		CONFIG_STATE_INIT,
		CONFIG_STATE_READ,
		CONFIG_STATE_WRITE,
		CONFIG_STATE_READY
		);
	RegistrationStatusType : {REDUND_UNREPLICABLE} 	STRUCT
		ActualMarkPosition : {REDUND_UNREPLICABLE} LREAL;
		MarkPositionError : {REDUND_UNREPLICABLE} LREAL;
		ActualProductLength : {REDUND_UNREPLICABLE} LREAL;
		ActualIntervalLength : {REDUND_UNREPLICABLE} LREAL;
		PhaseShift : {REDUND_UNREPLICABLE} LREAL;
		LastValidMarks : {REDUND_UNREPLICABLE} UDINT;
		Configuration : {REDUND_UNREPLICABLE} MpRegMarkDetectionConfigType;
	END_STRUCT;
END_TYPE
```

- Program Logical/MachineControl/CrossCutter/UnitTests/CutterTest (ANSIC) (no source held here)

### Program Logical/MachineControl/Conveyor/Conveyor (IEC)

#### AxisControl.st - Init, cyclic, exit code
```iecst
(***********************************************************************************************************************
* Copyright: B&R Industrial Automation GmbH
* Description: This program implements an axis control
***********************************************************************************************************************)

PROGRAM _INIT

    ST_name(0, ADR(AxisControl.Status.TaskName), 0);
    RecipeInit;

    ConfigurationInit;

    MpAlarmXCoreFB.Enable := TRUE;

    MpAxisBasicFB.Enable := TRUE;

    AxisInit;
END_PROGRAM

PROGRAM _CYCLIC

    MpAxisBasicFB.MpLink := ADR(gAxisConveyor);
    MC_BR_CheckRestorePositionDataFB.Axis := ADR(gAxisConveyor);

    SimulationControl;
    AxisStateMachine;
    AxisCyclic;
    RecipeCyclic;

    MpAlarmXCoreFB.MpLink := ADR(gAlarmXCore_Conveyor);
    MpAlarmXCoreFB();

END_PROGRAM

PROGRAM _EXIT

    MpRecipeRegPar_Par.Enable := FALSE;
    MpRecipeRegPar_Par();

    MpRecipeRegPar_Cfg.Enable := FALSE;
    MpRecipeRegPar_Cfg();

    MpAxisBasicFB.Enable := FALSE;
    MpAxisBasicFB();

    MpAlarmXCoreFB.Enable := FALSE;
    MpAlarmXCoreFB();

END_PROGRAM
```

#### AxisControl.typ - Local data types
```iecst
TYPE
	AxisSettingsType : {REDUND_UNREPLICABLE} 	STRUCT
		AxisFeatures : {REDUND_UNREPLICABLE} ARRAY[0..2]OF STRING[255];
		DriveConfiguration : {REDUND_UNREPLICABLE} McCfgPureVAxType;
		BaseConfiguration : {REDUND_UNREPLICABLE} McCfgAxType;
	END_STRUCT;
	AxisMachineSettingsType : {REDUND_UNREPLICABLE} 	STRUCT
		ReferencePosition : {REDUND_UNREPLICABLE} LREAL := 0; (*[mm] Axis position after reference*)
	END_STRUCT;
	AxisControlCommandType : {REDUND_UNREPLICABLE} 	STRUCT
		UpdatePreviewParameters : {REDUND_UNREPLICABLE} BOOL;
		LoadRecipeParameters : {REDUND_UNREPLICABLE} BOOL;
		SaveRecipeParameters : {REDUND_UNREPLICABLE} BOOL;
		Power : {REDUND_UNREPLICABLE} BOOL;
		Reference : {REDUND_UNREPLICABLE} BOOL;
		MoveAbsolute : {REDUND_UNREPLICABLE} BOOL;
		MoveAdditive : {REDUND_UNREPLICABLE} BOOL;
		MoveToStart : {REDUND_UNREPLICABLE} BOOL;
		Abort : {REDUND_UNREPLICABLE} BOOL;
		Stop : {REDUND_UNREPLICABLE} BOOL;
		Reset : {REDUND_UNREPLICABLE} BOOL;
		JogPositive : {REDUND_UNREPLICABLE} BOOL;
		JogNegative : {REDUND_UNREPLICABLE} BOOL;
		Start : {REDUND_UNREPLICABLE} BOOL;
	END_STRUCT;
	AxisControlParametersType : {REDUND_UNREPLICABLE} 	STRUCT
		HomePosition : {REDUND_UNREPLICABLE} LREAL := 0;
		Position : {REDUND_UNREPLICABLE} LREAL := 0;
		Distance : {REDUND_UNREPLICABLE} LREAL := 180;
		Velocity : {REDUND_UNREPLICABLE} REAL := 360;
		Acceleration : {REDUND_UNREPLICABLE} REAL := 360;
		Deceleration : {REDUND_UNREPLICABLE} REAL := 360;
		JogVelocity : {REDUND_UNREPLICABLE} REAL := 100;
		StopDeceleration : {REDUND_UNREPLICABLE} REAL := 720; (*[mm/s2] Deceleration for stopping*)
		ProductNumber : {REDUND_UNREPLICABLE} INT := 0; (*Product Number*)
		ProductLength : {REDUND_UNREPLICABLE} REAL := 70; (*Real Product Length*)
	END_STRUCT;
	AxisControlStatusType : {REDUND_UNREPLICABLE} 	STRUCT
		TaskName : {REDUND_UNREPLICABLE} STRING[80];
		MachineSettingsName : {REDUND_UNREPLICABLE} STRING[255];
		ProductSettingsName : {REDUND_UNREPLICABLE} STRING[255];
		ProductPreviewSettingsName : {REDUND_UNREPLICABLE} STRING[255];
		Status : {REDUND_UNREPLICABLE} STRING[80]; (*Machine Status*)
		IsReady : {REDUND_UNREPLICABLE} BOOL;
		ErrorActive : {REDUND_UNREPLICABLE} BOOL;
		Busy : {REDUND_UNREPLICABLE} BOOL;
		ReferenceRequired : {REDUND_UNREPLICABLE} BOOL;
		Position : {REDUND_UNREPLICABLE} LREAL;
		Velocity : {REDUND_UNREPLICABLE} REAL;
		Current : {REDUND_UNREPLICABLE} REAL;
		LagError : {REDUND_UNREPLICABLE} LREAL;
		MotorTemperature : {REDUND_UNREPLICABLE} REAL;
		IsHomed : {REDUND_UNREPLICABLE} BOOL;
		IsPowered : {REDUND_UNREPLICABLE} BOOL;
	END_STRUCT;
	AxisControlType : {REDUND_UNREPLICABLE} 	STRUCT
		Command : {REDUND_UNREPLICABLE} AxisControlCommandType;
		Parameters : {REDUND_UNREPLICABLE} AxisControlParametersType;
		Status : {REDUND_UNREPLICABLE} AxisControlStatusType;
	END_STRUCT;
	stateEnum :
		(
		STATE_INIT,
		STATE_POWER_ON,
		STATE_HOME,
		STATE_REFERENCE,
		STATE_MOVE_TO_HOME_POSITION,
		STATE_READY,
		STATE_MANUAL_OPERATION,
		STATE_AUTOMATIC_OPERATION,
		STATE_STOPPING,
		STATE_STOPPED,
		STATE_ABORTING,
		STATE_ABORTED,
		STATE_CLEARING,
		STATE_RESETTING
		);
	configurationStateEnum :
		(
		CONFIG_STATE_INIT,
		CONFIG_STATE_READ,
		CONFIG_STATE_WRITE,
		CONFIG_STATE_READY
		);
	automaticStateEnum :
		(
		AUTOMATIC_STATE_IDLE,
		AUTOMATIC_STATE_RUNNING
		);
	manualStateEnum :
		(
		MANUAL_STATE_IDLE,
		MANUAL_STATE_JOG,
		MANUAL_STATE_MOVE,
		MANUAL_STATE_STOPPING
		);
END_TYPE
```

- AxisControl.var (reference to Logical/Infrastructure/AxisTemplate/AxisControl/AxisControl.var)

#### SimulationControl.st
```iecst
ACTION SimulationControl:

	IF NOT (DiagCpuIsARsim() OR DiagCpuIsSimulated()) THEN
		RETURN;
    END_IF

//    IF ((MpAxisBasicFB.Info.ReadyToPowerOn = TRUE) AND (MpAxisBasicFB.PowerOn = FALSE)) THEN
//        AxisControl.Command.Power := TRUE;
//    END_IF

    IF ((MpAxisBasicFB.IsHomed = FALSE) AND (MpAxisBasicFB.Home = FALSE)) THEN
        AxisControl.Command.Reference := TRUE;
    END_IF

END_ACTION
```

#### AxisControlModes.st
```iecst
ACTION AxisInit:

END_ACTION

ACTION AxisCyclic:

    MpAlarmXControlSpeedNotSetFB.MpLink := ADR(gAlarmXCore_Conveyor);
    MpAlarmXControlSpeedNotSetFB.Enable := TRUE;
    MpAlarmXControlSpeedNotSetFB.Name := ADR('ConveyorSpeedNotSet');
    MpAlarmXControlSpeedNotSetFB();
    MpAlarmXControlSpeedNotSetFB.Reset := FALSE;

END_ACTION

ACTION AxisManual:

    MpAxisParameters.Jog.Velocity := AxisControl.Parameters.JogVelocity;
    MpAxisParameters.Position := AxisControl.Parameters.Position;
    MpAxisParameters.Distance := AxisControl.Parameters.Distance;
    MpAxisParameters.Acceleration := AxisControl.Parameters.Acceleration;
    MpAxisParameters.Deceleration := AxisControl.Parameters.Deceleration;

    CASE ManualState OF
        MANUAL_STATE_IDLE:
            IF ((AxisControl.Command.JogNegative = TRUE) OR (AxisControl.Command.JogPositive = TRUE)) THEN
                ManualState := MANUAL_STATE_JOG;
            ELSIF ((AxisControl.Command.MoveAbsolute = TRUE) OR (AxisControl.Command.MoveAdditive = TRUE)) THEN
                MpAxisBasicFB.MoveAbsolute := AxisControl.Command.MoveAbsolute;
                MpAxisBasicFB.MoveAdditive := AxisControl.Command.MoveAdditive;
                AxisControl.Command.MoveAbsolute := FALSE;
                AxisControl.Command.MoveAdditive := FALSE;
                ManualState := MANUAL_STATE_MOVE;
            END_IF

        MANUAL_STATE_JOG:
            MpAxisBasicFB.JogNegative := AxisControl.Command.JogNegative;
            MpAxisBasicFB.JogPositive := AxisControl.Command.JogPositive;
            IF (AxisControl.Command.Stop = TRUE) THEN
                AxisControl.Command.Stop := FALSE;
                MpAxisBasicFB.Stop := TRUE;
                ManualState := MANUAL_STATE_STOPPING;
            ELSIF ((AxisControl.Command.JogNegative = FALSE) AND (AxisControl.Command.JogPositive = FALSE)) THEN
                MpAxisBasicFB.Stop := FALSE;
                MpAxisBasicFB.JogPositive := FALSE;
                MpAxisBasicFB.JogNegative := FALSE;
                ManualState := MANUAL_STATE_STOPPING;
            END_IF

        MANUAL_STATE_MOVE:
            IF (AxisControl.Command.Stop = TRUE) THEN
                MpAxisBasicFB.MoveAbsolute := FALSE;
                MpAxisBasicFB.MoveAdditive := FALSE;
                AxisControl.Command.Stop := FALSE;
                MpAxisBasicFB.Stop := TRUE;
                ManualState := MANUAL_STATE_STOPPING;
            ELSIF (InPositionEdgePos.Q = TRUE) THEN
                MpAxisBasicFB.MoveAbsolute := FALSE;
                MpAxisBasicFB.MoveAdditive := FALSE;
                ManualState := MANUAL_STATE_IDLE;
                state := STATE_READY;
            ELSIF ((AxisControl.Command.JogNegative = TRUE) OR (AxisControl.Command.JogPositive = TRUE)) THEN
                MpAxisBasicFB.MoveAbsolute := FALSE;
                MpAxisBasicFB.MoveAdditive := FALSE;
                ManualState := MANUAL_STATE_JOG;
            END_IF

        MANUAL_STATE_STOPPING:
            MpAxisBasicFB.JogNegative := FALSE;
            MpAxisBasicFB.JogPositive := FALSE;
            MpAxisBasicFB.MoveAbsolute := FALSE;
            MpAxisBasicFB.MoveAdditive := FALSE;

            IF (MpAxisBasicFB.MoveActive = FALSE) THEN
                ManualState := MANUAL_STATE_IDLE;
                state := STATE_READY;
            END_IF
    END_CASE

END_ACTION

ACTION AxisAutomatic:

    CASE AutomaticState OF
        AUTOMATIC_STATE_IDLE:
            IF (AxisControl.Command.Start = TRUE) THEN
                MpAlarmXControlSpeedNotSetFB.Set := (MpAxisParameters.Velocity = 0);
                AxisControl.Command.Start := FALSE;
                AutomaticState := AUTOMATIC_STATE_RUNNING;
            END_IF

        AUTOMATIC_STATE_RUNNING:
            MpAxisBasicFB.MoveVelocity := TRUE;
            MpAxisParameters.Velocity := AxisControl.Parameters.Velocity;
            MpAxisParameters.Acceleration := AxisControl.Parameters.Acceleration;
            MpAxisParameters.Deceleration := AxisControl.Parameters.Deceleration;

            IF (AxisControl.Command.Stop = TRUE) THEN
                AxisControl.Command.Stop := FALSE;
                MpAxisBasicFB.MoveVelocity := FALSE;
                state := STATE_READY;
                AutomaticState := AUTOMATIC_STATE_IDLE;
            END_IF
    END_CASE

END_ACTION

ACTION AxisReset:

//    edge alarms don't require a reset
//    IF (MpAlarmXControlSpeedNotSetFB.Set = TRUE) THEN
//        MpAlarmXControlSpeedNotSetFB.Set := FALSE;
//        MpAlarmXControlSpeedNotSetFB.ID := MpAlarmXControlSpeedNotSetFB.InstanceID;
//        MpAlarmXControlSpeedNotSetFB.Reset := TRUE;
//    END_IF

END_ACTION
```

- AxisStateMachine.st (reference to Logical/Infrastructure/AxisTemplate/AxisControl/AxisStateMachine.st)

- ChangeConfiguration.st (reference to Logical/Infrastructure/AxisTemplate/AxisControl/ChangeConfiguration.st)

#### AutomaticCommand.st
```iecst
(* Returns True if an automatic command is active *)
FUNCTION AutomaticCommand

    AutomaticCommand := Commands.Start;

END_FUNCTION
```

- Recipe.st (reference to Logical/Infrastructure/AxisTemplate/AxisControl/Recipe.st)

#### Types.typ - not listed in the package file held
```iecst
TYPE
	AxisMachineSettingsType : {REDUND_UNREPLICABLE} 	STRUCT
		ReferencePosition : {REDUND_UNREPLICABLE} LREAL := 0; (*[mm] Axis position after reference*)
		AxisFeatures : {REDUND_UNREPLICABLE} ARRAY[0..2]OF STRING[255] := ['CamAut_cutting','ValueSource',''];
		DriveConfiguration : {REDUND_UNREPLICABLE} McCfgPureVAxType;
		BaseConfiguration : {REDUND_UNREPLICABLE} McCfgAxType;
	END_STRUCT;
	AxisControlCommandType : {REDUND_UNREPLICABLE} 	STRUCT
		UpdatePreviewParameters : {REDUND_UNREPLICABLE} BOOL;
		ResetEditParameters : {REDUND_UNREPLICABLE} BOOL;
		Power : {REDUND_UNREPLICABLE} BOOL;
		Reference : {REDUND_UNREPLICABLE} BOOL;
		MoveAbsolute : {REDUND_UNREPLICABLE} BOOL;
		MoveAdditive : {REDUND_UNREPLICABLE} BOOL;
		MoveToStart : {REDUND_UNREPLICABLE} BOOL;
		Abort : {REDUND_UNREPLICABLE} BOOL;
		Stop : {REDUND_UNREPLICABLE} BOOL;
		Reset : {REDUND_UNREPLICABLE} BOOL;
		JogPositive : {REDUND_UNREPLICABLE} BOOL;
		JogNegative : {REDUND_UNREPLICABLE} BOOL;
		Start : {REDUND_UNREPLICABLE} BOOL;
	END_STRUCT;
	AxisControlParametersType : {REDUND_UNREPLICABLE} 	STRUCT
		HomePosition : {REDUND_UNREPLICABLE} LREAL := 0;
		Position : {REDUND_UNREPLICABLE} LREAL := 0;
		Distance : {REDUND_UNREPLICABLE} LREAL := 180;
		Velocity : {REDUND_UNREPLICABLE} REAL := 360;
		Acceleration : {REDUND_UNREPLICABLE} REAL := 360;
		Deceleration : {REDUND_UNREPLICABLE} REAL := 360;
		JogVelocity : {REDUND_UNREPLICABLE} REAL := 100;
		StopDeceleration : {REDUND_UNREPLICABLE} REAL := 720; (*[mm/s2] Deceleration for stopping*)
		ProductNumber : {REDUND_UNREPLICABLE} INT := 0; (*Product Number*)
		ProductLength : {REDUND_UNREPLICABLE} REAL := 70; (*Real Product Length*)
	END_STRUCT;
	AxisControlStatusType : {REDUND_UNREPLICABLE} 	STRUCT
		TaskName : {REDUND_UNREPLICABLE} STRING[80];
		MachineSettingsName : {REDUND_UNREPLICABLE} STRING[255];
		ProductSettingsName : {REDUND_UNREPLICABLE} STRING[255];
		ProductPreviewSettingsName : {REDUND_UNREPLICABLE} STRING[255];
		Status : {REDUND_UNREPLICABLE} STRING[80]; (*Machine Status*)
		IsReady : {REDUND_UNREPLICABLE} BOOL;
		ErrorActive : {REDUND_UNREPLICABLE} BOOL;
		Busy : {REDUND_UNREPLICABLE} BOOL;
		ReferenceRequired : {REDUND_UNREPLICABLE} BOOL;
		Position : {REDUND_UNREPLICABLE} LREAL;
		Velocity : {REDUND_UNREPLICABLE} REAL;
		Current : {REDUND_UNREPLICABLE} REAL;
		LagError : {REDUND_UNREPLICABLE} LREAL;
		MotorTemperature : {REDUND_UNREPLICABLE} REAL;
		IsHomed : {REDUND_UNREPLICABLE} BOOL;
		IsPowered : {REDUND_UNREPLICABLE} BOOL;
	END_STRUCT;
	AxisControlType : {REDUND_UNREPLICABLE} 	STRUCT
		Command : {REDUND_UNREPLICABLE} AxisControlCommandType;
		Parameters : {REDUND_UNREPLICABLE} AxisControlParametersType;
		Status : {REDUND_UNREPLICABLE} AxisControlStatusType;
	END_STRUCT;
	stateEnum :
		(
		STATE_INIT,
		STATE_POWER_ON,
		STATE_HOME,
		STATE_REFERENCE,
		STATE_MOVE_TO_HOME_POSITION,
		STATE_READY,
		STATE_MANUAL_OPERATION,
		STATE_AUTOMATIC_OPERATION,
		STATE_STOPPING,
		STATE_STOPPED,
		STATE_ABORTING,
		STATE_ABORTED,
		STATE_CLEARING,
		STATE_RESETTING
		);
	configurationStateEnum :
		(
		CONFIG_STATE_INIT,
		CONFIG_STATE_READ,
		CONFIG_STATE_WRITE,
		CONFIG_STATE_READY
		);
	manualStateEnum :
		(
		MANUAL_STATE_IDLE,
		MANUAL_STATE_JOG,
		MANUAL_STATE_MOVE,
		MANUAL_STATE_STOPPING
		);
END_TYPE
```

### Package Logical/MachineControl/Conveyor/UnitTests - Multiple variants of valid test sets

### Program Logical/MachineControl/Conveyor/UnitTests/ConvTest (ANSIC) - Prototype for unit tests

- AxisControl.typ (reference to Logical/Infrastructure/AxisTemplate/AxisControl/AxisControl.typ)

- Visualisation Logical/mappView (not shown)

### Package Logical/UserPartition - User partition contents for mapp Framework

### Package Logical/UserPartition/Recipe - User partition files for mapp Recipe Framework

- Machine.mcfg - Default machine configuration file, XML format (not shown)

### Package Logical/UserPartition/Recipe/CSVformat - Container for CSV default files (same names as XML files) 

- Machine.mcfg - Default machine configuration file, CSV format (not shown)
